(* IEC 61131-3 sources: volt/packages/volt-lsp-iec/test-corpus/pro2193/Device/Plc Logic/Application/09 Misc/Library Manager/L_MC1P_MotionControlBasic (part 4) *)

(* ---- L_MC1P_DRIVESCALING_ENCI900.pou ---- *)
FUNCTION_BLOCK L_MC1P_DRIVESCALING_ENCI900 EXTENDS L_Mc1P_DriveScaling
END_FUNCTION_BLOCK

METHOD CALCACCFACTOR : BOOL
VAR_OUTPUT
	LRSCALEUNITTOACC : LREAL;
	LRSCALEACCTOUNIT : LREAL;
END_VAR
VAR_IN_OUT
	AXIS : _AXIS_REF_REAL;
END_VAR
END_METHOD

METHOD CALCSPEEDFACTOR : BOOL
VAR_OUTPUT
	LRSCALEUNITTOSPEED : LREAL;
	LRSCALESPEEDTOUNIT : LREAL;
END_VAR
VAR_IN_OUT
	AXIS : _AXIS_REF_REAL;
END_VAR
END_METHOD

METHOD CHECKVALIDPOSRESOLUTION : BOOL
VAR_INPUT
	DWPOSRESOLUTION : DWORD;
END_VAR
END_METHOD

METHOD POSDIFFTOSPEEDINC : DINT
VAR_INPUT
	DIPOSDIFF : DINT := 0;
	DWFACTOR : DWORD := 1000;
END_VAR
VAR_IN_OUT
	AXIS : _AXIS_REF_REAL;
END_VAR
END_METHOD

METHOD SPEEDTOPOSDIFFINC : DINT
VAR_INPUT
	DISPEED : DINT := 0;
	DWFACTOR : DWORD := 1000;
END_VAR
VAR_IN_OUT
	AXIS : _AXIS_REF_REAL;
	DIRES : DINT;
END_VAR
END_METHOD

(* ---- L_MC1P_DRIVESCALING_GENERICDRIVE.pou ---- *)
FUNCTION_BLOCK L_MC1P_DRIVESCALING_GENERICDRIVE
VAR_INPUT
	ITFGENERICCONFIG : L_MC1P_IGenericAxisConfiguration;
END_VAR
VAR
	PGENERICAXISCONFIGURATION : POINTER TO L_MC1P_GenericAxisConfiguration;
END_VAR
END_FUNCTION_BLOCK

METHOD CALCACCFACTOR : BOOL
VAR_OUTPUT
	LRSCALEUNITTOACC : LREAL;
	LRSCALEACCTOUNIT : LREAL;
END_VAR
VAR_IN_OUT
	AXIS : _AXIS_REF_REAL;
END_VAR
END_METHOD

METHOD CALCSPEEDFACTOR : BOOL
VAR_OUTPUT
	LRSCALEUNITTOSPEED : LREAL;
	LRSCALESPEEDTOUNIT : LREAL;
END_VAR
VAR_IN_OUT
	AXIS : _AXIS_REF_REAL;
END_VAR
END_METHOD

METHOD CALCTORQUEFACTOR : BOOL
VAR_OUTPUT
	LRSCALETORQUETONORM : LREAL;
	LRSCALETORQUETONORM2 : LREAL;
	LRSCALENORMTOTORQUE : LREAL;
END_VAR
VAR_IN_OUT
	AXIS : _AXIS_REF_REAL;
END_VAR
END_METHOD

METHOD CHECKVALIDPOSRESOLUTION : BOOL
VAR_INPUT
	DWPOSRESOLUTION : DWORD;
END_VAR
END_METHOD

METHOD GETDEFAULTTORQUE : LREAL
VAR_INPUT
	LRREFTORQUE : LREAL;
END_VAR
END_METHOD

METHOD POSDIFFTOSPEEDINC : DINT
VAR_INPUT
	DIPOSDIFF : DINT := 0;
	DWFACTOR : DWORD := 1000;
END_VAR
VAR_IN_OUT
	AXIS : _AXIS_REF_REAL;
END_VAR
END_METHOD

METHOD SPEEDTOPOSDIFFINC : DINT
VAR_INPUT
	DISPEED : DINT := 0;
	DWFACTOR : DWORD := 1000;
END_VAR
VAR_IN_OUT
	AXIS : _AXIS_REF_REAL;
	DIRES : DINT;
END_VAR
END_METHOD

METHOD UPDATEINTERFACE : BOOL
END_METHOD

(* ---- L_MC1P_DRIVESCALING_I500.pou ---- *)
FUNCTION_BLOCK L_MC1P_DRIVESCALING_I500 EXTENDS L_MC1P_DriveScaling
END_FUNCTION_BLOCK

METHOD CALCTORQUEFACTOR : BOOL
VAR_OUTPUT
	LRSCALETORQUETONORM : LREAL;
	LRSCALETORQUETONORM2 : LREAL;
	LRSCALENORMTOTORQUE : LREAL;
END_VAR
VAR_IN_OUT
	AXIS : _AXIS_REF_REAL;
END_VAR
END_METHOD

METHOD GETDEFAULTTORQUE : LREAL
VAR_INPUT
	LRREFTORQUE : LREAL;
END_VAR
END_METHOD

(* ---- L_MC1P_DRIVESCALING_I7XX.pou ---- *)
FUNCTION_BLOCK L_MC1P_DRIVESCALING_I7XX
END_FUNCTION_BLOCK

METHOD CALCACCFACTOR : BOOL
VAR_OUTPUT
	LRSCALEUNITTOACC : LREAL;
	LRSCALEACCTOUNIT : LREAL;
END_VAR
VAR_IN_OUT
	AXIS : _AXIS_REF_REAL;
END_VAR
END_METHOD

METHOD CALCSPEEDFACTOR : BOOL
VAR_OUTPUT
	LRSCALEUNITTOSPEED : LREAL;
	LRSCALESPEEDTOUNIT : LREAL;
END_VAR
VAR_IN_OUT
	AXIS : _AXIS_REF_REAL;
END_VAR
END_METHOD

METHOD CALCTORQUEFACTOR : BOOL
VAR_OUTPUT
	LRSCALETORQUETONORM : LREAL;
	LRSCALETORQUETONORM2 : LREAL;
	LRSCALENORMTOTORQUE : LREAL;
END_VAR
VAR_IN_OUT
	AXIS : _AXIS_REF_REAL;
END_VAR
END_METHOD

METHOD CHECKVALIDPOSRESOLUTION : BOOL
VAR_INPUT
	DWPOSRESOLUTION : DWORD;
END_VAR
END_METHOD

METHOD GETDEFAULTTORQUE : LREAL
VAR_INPUT
	LRREFTORQUE : LREAL;
END_VAR
END_METHOD

METHOD POSDIFFTOSPEEDINC : DINT
VAR_INPUT
	DIPOSDIFF : DINT := 0;
	DWFACTOR : DWORD := 1000;
END_VAR
VAR_IN_OUT
	AXIS : _AXIS_REF_REAL;
END_VAR
END_METHOD

METHOD SPEEDTOPOSDIFFINC : DINT
VAR_INPUT
	DISPEED : DINT := 0;
	DWFACTOR : DWORD := 1000;
END_VAR
VAR_IN_OUT
	AXIS : _AXIS_REF_REAL;
	DIRES : DINT;
END_VAR
END_METHOD

(* ---- L_MC1P_DRIVESPECIFIC_9400HL.pou ---- *)
FUNCTION_BLOCK L_MC1P_DRIVESPECIFIC_9400HL EXTENDS L_MC1P_DriveSpecific_CiA402
VAR
	TPWORKER : L_MC1P_TpWorker_CiA402;
	WSTATESM : WORD;
	DRIVEHOMESTATUSCHANGED : BOOL;
END_VAR
END_FUNCTION_BLOCK

METHOD CALCAFTERREADINPUTS
VAR_IN_OUT
	AXIS : _AXIS_REF_REAL;
END_VAR
END_METHOD

METHOD CALCBEFOREWRITEOUTPUTS
VAR_IN_OUT
	AXIS : _AXIS_REF_REAL;
END_VAR
END_METHOD

METHOD CHECKRESETHOMEPOS
VAR_INPUT
	WFDBSTATUSWORD : WORD;
END_VAR
VAR_IN_OUT
	AXIS : _AXIS_REF_REAL;
END_VAR
END_METHOD

METHOD GETADDITIONALSTATEINFOS : BOOL
VAR_IN_OUT
	AXIS : _AXIS_REF_REAL;
	SCSTATEINFO : L_MC1P_DriveStateCollection;
END_VAR
END_METHOD

METHOD GETCAUSEOFCINH : WORD
VAR_IN_OUT
	AXIS : _AXIS_REF_REAL;
END_VAR
END_METHOD

METHOD GETRECEIVEDATAIMPL : DWORD
VAR_INPUT
	LWMASK : LWORD;
END_VAR
VAR_IN_OUT
	AXIS : _AXIS_REF_REAL;
END_VAR
END_METHOD

METHOD GETSTOACTIVEFROMSTATE : BOOL
VAR_IN_OUT
	AXIS : _AXIS_REF_REAL;
END_VAR
END_METHOD

METHOD HOMECONFIG : BOOL
VAR_INPUT
	LRPOSITION : LREAL;
END_VAR
VAR_OUTPUT
	WINDEX : WORD;
	BYSUBINDEX : BYTE;
	BYNROFBYTE : BYTE;
	DWDATA : DWORD;
	XWRITEPARAM : BOOL;
	XDONE : BOOL;
	XERROR : BOOL;
END_VAR
VAR_IN_OUT
	AXIS : _AXIS_REF_REAL;
	SCHOMEDATA : L_MC1P_HomeParameter;
	WSTEP : WORD;
END_VAR
END_METHOD

METHOD PROZESSCONTROLWORD : BOOL
VAR_IN_OUT
	AXIS : _AXIS_REF_REAL;
END_VAR
END_METHOD

METHOD RECEIVEPARAMETERCALC
VAR_IN_OUT
	AXIS : _AXIS_REF_REAL;
	DATA : ARRAY [1..L_MC1P_Constants.gc_Rec_MaxDataIndex] OF POINTER TO L_MC1P_MappedElement;
END_VAR
END_METHOD

METHOD SETAXISPROPERTIES
VAR_IN_OUT
	AXIS : _AXIS_REF_REAL;
	AXISPROPERTIES : L_MC1P_AxisProperties;
END_VAR
END_METHOD

METHOD SETAXISSTATUSWORD
VAR_IN_OUT
	AXIS : _AXIS_REF_REAL;
	DWAXISSTATUS : DWORD;
END_VAR
END_METHOD

METHOD SETDRIVECONFIGINIT
VAR_IN_OUT
	AXIS : _AXIS_REF_REAL;
END_VAR
END_METHOD

METHOD TRANSMITPARAMETERCALC
VAR_IN_OUT
	AXIS : _AXIS_REF_REAL;
	DATA : ARRAY [1..L_MC1P_Constants.gc_Trans_MaxDataIndex] OF POINTER TO L_MC1P_MappedElement;
END_VAR
END_METHOD

(* ---- L_MC1P_DRIVESPECIFIC_BASIC.pou ---- *)
FUNCTION_BLOCK L_MC1P_DRIVESPECIFIC_BASIC
VAR_INPUT
	XDEFAULTBEHAVIOURASVIRTUAL : BOOL := FALSE;
END_VAR
VAR
	XENABLE : BOOL;
	DIPOS : DINT;
	DIVEL : DINT;
	ITORQUE : INT;
	ITORQUELIMPOS : INT;
	ITORQUELIMNEG : INT;
	DIFOLLOWINGERROR : DINT;
	WERRORCODE : WORD;
	BASICINITERROR : L_IE1P_Error;
	DRIVEHOMESTATUSCHANGED : BOOL;
	DRIVEINITIALIZED : BOOL;
	DRIVEINITIALIZEDERRORREASON : L_IE1P_Error;
	GETITFBRAKE : L_MC1P_IAXIS_REF_BRAKE;
	GETITFCMDBRAKEGRINDIN : L_MC1P_IAxisCommmand;
	GETITFCMDBRAKETEST : L_MC1P_IAxisCommmand;
	HOMESEQUENCESTATE : WORD;
	ITFMOLACCESS : L_MC1P_IMOLAccess;
	ITFPLIACCESS : L_MC1P_IPLIAccess;
	PINSTANCE : POINTER TO BYTE;
END_VAR
END_FUNCTION_BLOCK

METHOD CALCAFTERREADINPUTS
VAR_IN_OUT
	AXIS : _AXIS_REF_REAL;
END_VAR
END_METHOD

METHOD CALCBEFOREREADINPUTS
VAR_IN_OUT
	AXIS : _AXIS_REF_REAL;
END_VAR
END_METHOD

METHOD CALCBEFOREWRITEOUTPUTS
VAR_IN_OUT
	AXIS : _AXIS_REF_REAL;
END_VAR
END_METHOD

METHOD CHECKAVAILABLECONTROLMODE : BOOL
VAR_IN_OUT
	AXIS : _AXIS_REF_REAL;
	POSCTRLDRIVEAVAILABLE : L_IE1P_Error;
	POSCTRLPLCAVAILABLE : L_IE1P_Error;
	SPEEDCTRLDRIVEAVAILABLE : L_IE1P_Error;
	TORQUECTRLDRIVE : L_IE1P_Error;
END_VAR
END_METHOD

METHOD CHECKRESETHOMEPOS
VAR_INPUT
	WFDBSTATUSWORD : WORD;
END_VAR
VAR_IN_OUT
	AXIS : _AXIS_REF_REAL;
END_VAR
END_METHOD

METHOD CHECKSAFETYOPTIONAVAILABLE : BOOL
VAR_INPUT
	DWPRODUCTCODE : DWORD;
END_VAR
END_METHOD

METHOD COLLECTDRIVESTATE : BOOL
VAR_IN_OUT
	AXIS : _AXIS_REF_REAL;
	SCSTATEINFO : L_MC1P_DriveStateCollection;
END_VAR
END_METHOD

METHOD CONTROLDRIVE : BOOL
VAR_INPUT
	XENABLE : BOOL;
END_VAR
VAR_IN_OUT
	AXIS : _AXIS_REF_REAL;
END_VAR
END_METHOD

METHOD DRIVECONFIGDATA
VAR_INPUT
	PCONFIGINFO : POINTER TO L_MC1P_AdditionalConfigInfo;
END_VAR
VAR_IN_OUT
	AXIS : _AXIS_REF_REAL;
END_VAR
END_METHOD

METHOD DRIVEFAULTSTATUS : BOOL
VAR_IN_OUT
	AXIS : _AXIS_REF_REAL;
	SCSTATEINFO : L_MC1P_DriveStateCollection;
END_VAR
END_METHOD

METHOD GETBRAKE : POINTER TO L_MC1P_BrakeControlBase
VAR_IN_OUT
	AXIS : _AXIS_REF_REAL;
END_VAR
END_METHOD

METHOD GETBRAKESERVICE : POINTER TO L_MC1P_BrakeService
VAR_IN_OUT
	AXIS : _AXIS_REF_REAL;
END_VAR
END_METHOD

METHOD GETCAUSEOFCINH : WORD
VAR_IN_OUT
	AXIS : _AXIS_REF_REAL;
END_VAR
END_METHOD

METHOD GETFDBSTATUSWORD : WORD
VAR_IN_OUT
	AXIS : _AXIS_REF_REAL;
END_VAR
END_METHOD

METHOD GETIECADRESS : BOOL
VAR_IN_OUT
	AXIS : _AXIS_REF_REAL;
	M_PPDOINFOCONNECTOR : POINTER TO IoConfigConnector;
	ATRANSELEMENT : ARRAY [1.._AXIS_REF_REAL.c_wMaxTransElem] OF L_MC1P_MappedElement;
	WTRANSELEMENTS : WORD;
	LWTRANSDATA : LWORD;
	LWRECDATA : LWORD;
	WRECEIVEELEMENTS : WORD;
	ARECEIVEELEMENT : ARRAY [1.._AXIS_REF_REAL.c_wMaxRecElem] OF L_MC1P_MappedElement;
END_VAR
END_METHOD

METHOD GETOPTIONALACTVEL : BOOL
VAR_IN_OUT
	LRVEL : LREAL;
END_VAR
END_METHOD

METHOD GETRECEIVEDATAIMPL : DWORD
VAR_INPUT
	LWMASK : LWORD;
END_VAR
VAR_IN_OUT
	AXIS : _AXIS_REF_REAL;
END_VAR
END_METHOD

METHOD GETSTATUSWORDS
VAR_OUTPUT
	STATUSWORD1 : WORD;
	STATUSWORD2 : WORD;
	STATUSWORD3 : WORD;
	STATUSWORD4 : WORD;
END_VAR
VAR_IN_OUT
	AXIS : _AXIS_REF_REAL;
END_VAR
END_METHOD

METHOD GETTRANSMITDATAIMPL : DWORD
VAR_INPUT
	LWMASK : LWORD;
END_VAR
VAR_IN_OUT
	AXIS : _AXIS_REF_REAL;
END_VAR
END_METHOD

METHOD GETTRANSMITDATALREALIMPL : LREAL
VAR_INPUT
	LWMASK : LWORD;
END_VAR
VAR_IN_OUT
	AXIS : _AXIS_REF_REAL;
END_VAR
END_METHOD

METHOD HOMECONFIG : BOOL
VAR_INPUT
	LRPOSITION : LREAL;
END_VAR
VAR_OUTPUT
	WINDEX : WORD;
	BYSUBINDEX : BYTE;
	BYNROFBYTE : BYTE;
	DWDATA : DWORD;
	XWRITEPARAM : BOOL;
	XDONE : BOOL;
	XERROR : BOOL;
END_VAR
VAR_IN_OUT
	AXIS : _AXIS_REF_REAL;
	SCHOMEDATA : L_MC1P_HomeParameter;
	WSTEP : WORD;
END_VAR
END_METHOD

METHOD HOMEPOSPERMANENTSETACTIVE : BOOL
VAR_IN_OUT
	AXIS : _AXIS_REF_REAL;
END_VAR
END_METHOD

METHOD RECEIVEPARAMETER
VAR_INPUT
	WPARAMETER : WORD;
	PADRESS : POINTER TO BYTE;
	WSIZE : WORD;
END_VAR
VAR_IN_OUT
	AXIS : _AXIS_REF_REAL;
END_VAR
END_METHOD

METHOD RECEIVEPARAMETERCALC
VAR_IN_OUT
	AXIS : _AXIS_REF_REAL;
	DATA : ARRAY [1..L_MC1P_Constants.gc_Rec_MaxDataIndex] OF POINTER TO L_MC1P_MappedElement;
END_VAR
END_METHOD

METHOD RESETDRIVECONTROL
VAR_INPUT
	XRESETDRIVEERROR : BOOL;
END_VAR
END_METHOD

METHOD RESTOREADDITIONALRETAINDATA
VAR_INPUT
	PDATA : POINTER TO L_MC1P_uRetainData;
END_VAR
END_METHOD

METHOD SETAXISPROPERTIES
VAR_IN_OUT
	AXIS : _AXIS_REF_REAL;
	AXISPROPERTIES : L_MC1P_AxisProperties;
END_VAR
END_METHOD

METHOD SETAXISSTATUSWORD
VAR_IN_OUT
	AXIS : _AXIS_REF_REAL;
	DWAXISSTATUS : DWORD;
END_VAR
END_METHOD

METHOD SETBASICINITIALISATION
VAR_IN_OUT
	AXIS : _AXIS_REF_REAL;
END_VAR
END_METHOD

METHOD SETCONTROLWORDS
VAR_INPUT
	CONTROLWORD1 : WORD;
	CONTROLWORD2 : WORD;
	CONTROLWORD3 : WORD;
	CONTROLWORD4 : WORD;
END_VAR
VAR_IN_OUT
	AXIS : _AXIS_REF_REAL;
END_VAR
END_METHOD

METHOD SETDCBRAKE
VAR_INPUT
	XSETDCBRAKE : BOOL;
END_VAR
VAR_OUTPUT
	XDCBRAKEACTIVE : BOOL;
END_VAR
VAR_IN_OUT
	AXIS : _AXIS_REF_REAL;
END_VAR
END_METHOD

METHOD SETDRIVECONFIG
VAR_OUTPUT
	XDONE : BOOL;
	XERROR : BOOL;
	WERRORID : WORD;
END_VAR
VAR_IN_OUT
	AXIS : _AXIS_REF_REAL;
END_VAR
END_METHOD

METHOD SETDRIVECONFIGINIT
VAR_IN_OUT
	AXIS : _AXIS_REF_REAL;
END_VAR
END_METHOD

METHOD SETSPEEDCTRLLIMITATION : BOOL
VAR_INPUT
	XLIMIT : BOOL;
END_VAR
VAR_IN_OUT
	AXIS : _AXIS_REF_REAL;
END_VAR
END_METHOD

METHOD SETSPEEDCTRLLOADVALUE
VAR_INPUT
	XLOAD : BOOL;
	LRVALUE : LREAL;
END_VAR
VAR_IN_OUT
	AXIS : _AXIS_REF_REAL;
END_VAR
END_METHOD

METHOD STOREADDITIONALRETAINDATA
VAR_INPUT
	PDATA : POINTER TO L_MC1P_uRetainData;
END_VAR
END_METHOD

METHOD TRANSMITPARAMETER
VAR_INPUT
	WPARAMETER : WORD;
	PADRESS : POINTER TO BYTE;
	WSIZE : WORD;
END_VAR
VAR_IN_OUT
	AXIS : _AXIS_REF_REAL;
END_VAR
END_METHOD

METHOD TRANSMITPARAMETERCALC
VAR_IN_OUT
	AXIS : _AXIS_REF_REAL;
	DATA : ARRAY [1..L_MC1P_Constants.gc_Trans_MaxDataIndex] OF POINTER TO L_MC1P_MappedElement;
END_VAR
END_METHOD

METHOD UPDATEMAPPING
VAR_INPUT
	PTASKMAPLIST : POINTER TO IoStandard.IoConfigTaskMap;
	NCOUNT : DINT;
	PPDOINFOCONNECTOR : POINTER TO IoConfigConnector;
END_VAR
VAR_IN_OUT
	AXIS : _AXIS_REF_REAL;
END_VAR
END_METHOD

(* ---- L_MC1P_DRIVESPECIFIC_CIA402.pou ---- *)
FUNCTION_BLOCK L_MC1P_DRIVESPECIFIC_CIA402
VAR_INPUT
	WOFFSETDRIVEPARA : WORD;
END_VAR
VAR
	ECONTROLMODEDRIVE : SINT := 0;
	XUSEIPMODENOTCSP : BOOL := FALSE;
	XUSEVLMODENOTCSV : BOOL := FALSE;
	CIA_CTRL : WORD;
	CIA_OPMOD : SINT;
	CIA_STATE : WORD;
	CIA_OPMODACT : SINT;
	CIA_VLACTVELOCITY : INT;
	CIA_VLTARGETVELOCITY : INT;
	CIA_STATEOLD : WORD;
	WHOMESTATE : WORD;
	REFCIA_CTRL : REFERENCE TO WORD;
	REFCIA_OPMOD : REFERENCE TO SINT;
	REFCIA_STATE : REFERENCE TO WORD;
	REFCIA_OPMODACT : REFERENCE TO SINT;
	DWSAFETYCONTROL : DWORD;
	DWSAFETYSTATE : DWORD;
	DWSAFETYIOSTATE : DWORD;
	WLENZEEXTSTATUSWORD : WORD := 0;
	XTEXTREFID603FSUPPORTED : BOOL;
	WTEXTREFID603F : WORD;
	WTEXTREFID_SLAVE : WORD;
	LRDECTIME : LREAL;
	XQSPRAMPEND : BOOL;
	BASICINITERROR : L_IE1P_Types.L_IE1P_Error;
	DRIVEHOMESTATUSCHANGED : BOOL;
	DRIVEINITIALIZED : BOOL;
	DRIVEINITIALIZEDERRORREASON : L_IE1P_Types.L_IE1P_Error;
	GETITFBRAKE : L_MC1P_IAXIS_REF_BRAKE;
	GETITFCMDBRAKEGRINDIN : L_MC1P_IAxisCommmand;
	GETITFCMDBRAKETEST : L_MC1P_IAxisCommmand;
	HOMESEQUENCESTATE : WORD;
	ITFMOLACCESS : L_MC1P_IMOLAccess;
	ITFPLIACCESS : L_MC1P_IPLIAccess;
	PINSTANCE : POINTER TO BYTE;
END_VAR
END_FUNCTION_BLOCK

METHOD CALCAFTERCIA402STM : BOOL
VAR_IN_OUT
	AXIS : _AXIS_REF_REAL;
END_VAR
END_METHOD

METHOD GETADDITIONALSTATEINFOS : BOOL
VAR_IN_OUT
	AXIS : _AXIS_REF_REAL;
	SCSTATEINFO : L_MC1P_DriveStateCollection;
END_VAR
END_METHOD

METHOD GETDRIVEQSPDONE : BOOL
VAR_IN_OUT
	AXIS : _AXIS_REF_REAL;
	SCSTATEINFO : L_MC1P_DriveStateCollection;
END_VAR
END_METHOD

METHOD GETINTCONTROLMODE : SINT
VAR_INPUT
	ECONTROLMODE : L_MC1P_ControlMode;
END_VAR
VAR_IN_OUT
	AXIS : _AXIS_REF_REAL;
END_VAR
END_METHOD

METHOD GETSTOACTIVEFROMSTATE : BOOL
VAR_IN_OUT
	AXIS : _AXIS_REF_REAL;
END_VAR
END_METHOD

METHOD GETTEXTREFIDFROMERRORCODE : WORD
VAR_INPUT
	DWERRORID : DWORD;
END_VAR
VAR_IN_OUT
	AXIS : _AXIS_REF_REAL;
END_VAR
END_METHOD

METHOD GETTEXTREFIDFROMTABLE : BOOL
VAR_INPUT
	DWERRORID : DWORD;
	XSAFETYDEVICE : BOOL;
END_VAR
VAR_IN_OUT
	WTEXTREFID : WORD;
END_VAR
END_METHOD

METHOD HOMESEQUENCE
VAR_IN_OUT
	AXIS : _AXIS_REF_REAL;
END_VAR
END_METHOD

METHOD PROZESSCONTROLWORD : BOOL
VAR_IN_OUT
	AXIS : _AXIS_REF_REAL;
END_VAR
END_METHOD

METHOD SERVICEMODEHANDLINGINDRIVEACTIVE : BOOL
END_METHOD

METHOD FB_INIT : BOOL
VAR_INPUT
	BINITRETAINS : BOOL;
	BINCOPYCODE : BOOL;
END_VAR
END_METHOD

METHOD CALCAFTERREADINPUTS
VAR_IN_OUT
	AXIS : _AXIS_REF_REAL;
END_VAR
END_METHOD

METHOD CALCBEFOREREADINPUTS
VAR_IN_OUT
	AXIS : _AXIS_REF_REAL;
END_VAR
END_METHOD

METHOD CALCBEFOREWRITEOUTPUTS
VAR_IN_OUT
	AXIS : _AXIS_REF_REAL;
END_VAR
END_METHOD

METHOD CHECKAVAILABLECONTROLMODE : BOOL
VAR_IN_OUT
	AXIS : _AXIS_REF_REAL;
	POSCTRLDRIVEAVAILABLE : L_IE1P_Types.L_IE1P_Error;
	POSCTRLPLCAVAILABLE : L_IE1P_Types.L_IE1P_Error;
	SPEEDCTRLDRIVEAVAILABLE : L_IE1P_Types.L_IE1P_Error;
	TORQUECTRLDRIVE : L_IE1P_Types.L_IE1P_Error;
END_VAR
END_METHOD

METHOD CHECKRESETHOMEPOS
VAR_INPUT
	WFDBSTATUSWORD : WORD;
END_VAR
VAR_IN_OUT
	AXIS : _AXIS_REF_REAL;
END_VAR
END_METHOD

METHOD CHECKSAFETYOPTIONAVAILABLE : BOOL
VAR_INPUT
	DWPRODUCTCODE : DWORD;
END_VAR
END_METHOD

METHOD COLLECTDRIVESTATE : BOOL
VAR_IN_OUT
	AXIS : _AXIS_REF_REAL;
	SCSTATEINFO : L_MC1P_DriveStateCollection;
END_VAR
END_METHOD

METHOD CONTROLDRIVE : BOOL
VAR_INPUT
	XENABLE : BOOL;
END_VAR
VAR_IN_OUT
	AXIS : _AXIS_REF_REAL;
END_VAR
END_METHOD

METHOD DRIVECONFIGDATA
VAR_INPUT
	PCONFIGINFO : POINTER TO L_MC1P_AdditionalConfigInfo;
END_VAR
VAR_IN_OUT
	AXIS : _AXIS_REF_REAL;
END_VAR
END_METHOD

METHOD DRIVEFAULTSTATUS : BOOL
VAR_IN_OUT
	AXIS : _AXIS_REF_REAL;
	SCSTATEINFO : L_MC1P_DriveStateCollection;
END_VAR
END_METHOD

METHOD GETBRAKE : POINTER TO L_MC1P_BrakeControlBase
VAR_IN_OUT
	AXIS : _AXIS_REF_REAL;
END_VAR
END_METHOD

METHOD GETBRAKESERVICE : POINTER TO L_MC1P_BrakeService
VAR_IN_OUT
	AXIS : _AXIS_REF_REAL;
END_VAR
END_METHOD

METHOD GETCAUSEOFCINH : WORD
VAR_IN_OUT
	AXIS : _AXIS_REF_REAL;
END_VAR
END_METHOD

METHOD GETFDBSTATUSWORD : WORD
VAR_IN_OUT
	AXIS : _AXIS_REF_REAL;
END_VAR
END_METHOD

METHOD GETIECADRESS : BOOL
VAR_IN_OUT
	AXIS : _AXIS_REF_REAL;
	M_PPDOINFOCONNECTOR : POINTER TO IoStandard.IoConfigConnector;
	ATRANSELEMENT : ARRAY [1..._AXIS_REF_REAL.c_wMaxTransElem] OF L_MC1P_MappedElement;
	WTRANSELEMENTS : WORD;
	LWTRANSDATA : LWORD;
	LWRECDATA : LWORD;
	WRECEIVEELEMENTS : WORD;
	ARECEIVEELEMENT : ARRAY [1..._AXIS_REF_REAL.c_wMaxRecElem] OF L_MC1P_MappedElement;
END_VAR
END_METHOD

METHOD GETOPTIONALACTVEL : BOOL
VAR_IN_OUT
	LRVEL : LREAL;
END_VAR
END_METHOD

METHOD GETRECEIVEDATAIMPL : DWORD
VAR_INPUT
	LWMASK : LWORD;
END_VAR
VAR_IN_OUT
	AXIS : _AXIS_REF_REAL;
END_VAR
END_METHOD

METHOD GETSTATUSWORDS
VAR_OUTPUT
	STATUSWORD1 : WORD;
	STATUSWORD2 : WORD;
	STATUSWORD3 : WORD;
	STATUSWORD4 : WORD;
END_VAR
VAR_IN_OUT
	AXIS : _AXIS_REF_REAL;
END_VAR
END_METHOD

METHOD GETTRANSMITDATAIMPL : DWORD
VAR_INPUT
	LWMASK : LWORD;
END_VAR
VAR_IN_OUT
	AXIS : _AXIS_REF_REAL;
END_VAR
END_METHOD

METHOD GETTRANSMITDATALREALIMPL : LREAL
VAR_INPUT
	LWMASK : LWORD;
END_VAR
VAR_IN_OUT
	AXIS : _AXIS_REF_REAL;
END_VAR
END_METHOD

METHOD HOMECONFIG : BOOL
VAR_INPUT
	LRPOSITION : LREAL;
END_VAR
VAR_OUTPUT
	WINDEX : WORD;
	BYSUBINDEX : BYTE;
	BYNROFBYTE : BYTE;
	DWDATA : DWORD;
	XWRITEPARAM : BOOL;
	XDONE : BOOL;
	XERROR : BOOL;
END_VAR
VAR_IN_OUT
	AXIS : _AXIS_REF_REAL;
	SCHOMEDATA : L_MC1P_HomeParameter;
	WSTEP : WORD;
END_VAR
END_METHOD

METHOD HOMEPOSPERMANENTSETACTIVE : BOOL
VAR_IN_OUT
	AXIS : _AXIS_REF_REAL;
END_VAR
END_METHOD

METHOD RECEIVEPARAMETERCALC
VAR_IN_OUT
	AXIS : _AXIS_REF_REAL;
	DATA : ARRAY [1..L_MC1P_Constants.gc_Rec_MaxDataIndex] OF POINTER TO L_MC1P_MappedElement;
END_VAR
END_METHOD

METHOD RECEIVEPARAMETER
VAR_INPUT
	WPARAMETER : WORD;
	PADRESS : POINTER TO BYTE;
	WSIZE : WORD;
END_VAR
VAR_IN_OUT
	AXIS : _AXIS_REF_REAL;
END_VAR
END_METHOD

METHOD RESETDRIVECONTROL
VAR_INPUT
	XRESETDRIVEERROR : BOOL;
END_VAR
END_METHOD

METHOD RESTOREADDITIONALRETAINDATA
VAR_INPUT
	PDATA : POINTER TO L_MC1P_uRetainData;
END_VAR
END_METHOD

METHOD SETAXISPROPERTIES
VAR_IN_OUT
	AXIS : _AXIS_REF_REAL;
	AXISPROPERTIES : L_MC1P_AxisProperties;
END_VAR
END_METHOD

METHOD SETAXISSTATUSWORD
VAR_IN_OUT
	AXIS : _AXIS_REF_REAL;
	DWAXISSTATUS : DWORD;
END_VAR
END_METHOD

METHOD SETBASICINITIALISATION
VAR_IN_OUT
	AXIS : _AXIS_REF_REAL;
END_VAR
END_METHOD

METHOD SETCONTROLWORDS
VAR_INPUT
	CONTROLWORD1 : WORD;
	CONTROLWORD2 : WORD;
	CONTROLWORD3 : WORD;
	CONTROLWORD4 : WORD;
END_VAR
VAR_IN_OUT
	AXIS : _AXIS_REF_REAL;
END_VAR
END_METHOD

METHOD SETDCBRAKE
VAR_INPUT
	XSETDCBRAKE : BOOL;
END_VAR
VAR_OUTPUT
	XDCBRAKEACTIVE : BOOL;
END_VAR
VAR_IN_OUT
	AXIS : _AXIS_REF_REAL;
END_VAR
END_METHOD

METHOD SETDRIVECONFIGINIT
VAR_IN_OUT
	AXIS : _AXIS_REF_REAL;
END_VAR
END_METHOD

METHOD SETSPEEDCTRLLIMITATION : BOOL
VAR_INPUT
	XLIMIT : BOOL;
END_VAR
VAR_IN_OUT
	AXIS : _AXIS_REF_REAL;
END_VAR
END_METHOD

METHOD SETSPEEDCTRLLOADVALUE
VAR_INPUT
	XLOAD : BOOL;
	LRVALUE : LREAL;
END_VAR
VAR_IN_OUT
	AXIS : _AXIS_REF_REAL;
END_VAR
END_METHOD

METHOD STOREADDITIONALRETAINDATA
VAR_INPUT
	PDATA : POINTER TO L_MC1P_uRetainData;
END_VAR
END_METHOD

METHOD TRANSMITPARAMETERCALC
VAR_IN_OUT
	AXIS : _AXIS_REF_REAL;
	DATA : ARRAY [1..L_MC1P_Constants.gc_Trans_MaxDataIndex] OF POINTER TO L_MC1P_MappedElement;
END_VAR
END_METHOD

METHOD TRANSMITPARAMETER
VAR_INPUT
	WPARAMETER : WORD;
	PADRESS : POINTER TO BYTE;
	WSIZE : WORD;
END_VAR
VAR_IN_OUT
	AXIS : _AXIS_REF_REAL;
END_VAR
END_METHOD

METHOD UPDATEMAPPING
VAR_INPUT
	PTASKMAPLIST : POINTER TO IoStandard.IoConfigTaskMap;
	NCOUNT : DINT;
	PPDOINFOCONNECTOR : POINTER TO IoStandard.IoConfigConnector;
END_VAR
VAR_IN_OUT
	AXIS : _AXIS_REF_REAL;
END_VAR
END_METHOD

(* ---- L_MC1P_DRIVESPECIFIC_ENC.pou ---- *)
FUNCTION_BLOCK L_MC1P_DRIVESPECIFIC_ENC
VAR
	BASICINITERROR : L_IE1P_Error;
	DRIVEHOMESTATUSCHANGED : BOOL;
	DRIVEINITIALIZED : BOOL;
	DRIVEINITIALIZEDERRORREASON : L_IE1P_Error;
	GETITFBRAKE : L_MC1P_IAXIS_REF_BRAKE;
	GETITFCMDBRAKEGRINDIN : L_MC1P_IAxisCommmand;
	GETITFCMDBRAKETEST : L_MC1P_IAxisCommmand;
	HOMESEQUENCESTATE : WORD;
	ITFMOLACCESS : L_MC1P_IMOLAccess;
	ITFPLIACCESS : L_MC1P_IPLIAccess;
	PINSTANCE : POINTER TO BYTE;
END_VAR
END_FUNCTION_BLOCK

METHOD CALCAFTERREADINPUTS
VAR_IN_OUT
	AXIS : _AXIS_REF_REAL;
END_VAR
END_METHOD

METHOD CALCBEFOREREADINPUTS
VAR_IN_OUT
	AXIS : _AXIS_REF_REAL;
END_VAR
END_METHOD

METHOD CALCBEFOREWRITEOUTPUTS
VAR_IN_OUT
	AXIS : _AXIS_REF_REAL;
END_VAR
END_METHOD

METHOD CHECKAVAILABLECONTROLMODE : BOOL
VAR_IN_OUT
	AXIS : _AXIS_REF_REAL;
	POSCTRLDRIVEAVAILABLE : L_IE1P_Error;
	POSCTRLPLCAVAILABLE : L_IE1P_Error;
	SPEEDCTRLDRIVEAVAILABLE : L_IE1P_Error;
	TORQUECTRLDRIVE : L_IE1P_Error;
END_VAR
END_METHOD

METHOD CHECKRESETHOMEPOS
VAR_INPUT
	WFDBSTATUSWORD : WORD;
END_VAR
VAR_IN_OUT
	AXIS : _AXIS_REF_REAL;
END_VAR
END_METHOD

METHOD CHECKSAFETYOPTIONAVAILABLE : BOOL
VAR_INPUT
	DWPRODUCTCODE : DWORD;
END_VAR
END_METHOD

METHOD COLLECTDRIVESTATE : BOOL
VAR_IN_OUT
	AXIS : _AXIS_REF_REAL;
	SCSTATEINFO : L_MC1P_DriveStateCollection;
END_VAR
END_METHOD

METHOD CONTROLDRIVE : BOOL
VAR_INPUT
	XENABLE : BOOL;
END_VAR
VAR_IN_OUT
	AXIS : _AXIS_REF_REAL;
END_VAR
END_METHOD

METHOD DRIVECONFIGDATA
VAR_INPUT
	PCONFIGINFO : POINTER TO L_MC1P_AdditionalConfigInfo;
END_VAR
VAR_IN_OUT
	AXIS : _AXIS_REF_REAL;
END_VAR
END_METHOD

METHOD DRIVEFAULTSTATUS : BOOL
VAR_IN_OUT
	AXIS : _AXIS_REF_REAL;
	SCSTATEINFO : L_MC1P_DriveStateCollection;
END_VAR
END_METHOD

METHOD GETBRAKE : POINTER TO L_MC1P_BrakeControlBase
VAR_IN_OUT
	AXIS : _AXIS_REF_REAL;
END_VAR
END_METHOD

METHOD GETBRAKESERVICE : POINTER TO L_MC1P_BrakeService
VAR_IN_OUT
	AXIS : _AXIS_REF_REAL;
END_VAR
END_METHOD

METHOD GETCAUSEOFCINH : WORD
VAR_IN_OUT
	AXIS : _AXIS_REF_REAL;
END_VAR
END_METHOD

METHOD GETFDBSTATUSWORD : WORD
VAR_IN_OUT
	AXIS : _AXIS_REF_REAL;
END_VAR
END_METHOD

METHOD GETIECADRESS : BOOL
VAR_IN_OUT
	AXIS : _AXIS_REF_REAL;
	M_PPDOINFOCONNECTOR : POINTER TO IoConfigConnector;
	ATRANSELEMENT : ARRAY [1.._AXIS_REF_REAL.c_wMaxTransElem] OF L_MC1P_MappedElement;
	WTRANSELEMENTS : WORD;
	LWTRANSDATA : LWORD;
	LWRECDATA : LWORD;
	WRECEIVEELEMENTS : WORD;
	ARECEIVEELEMENT : ARRAY [1.._AXIS_REF_REAL.c_wMaxRecElem] OF L_MC1P_MappedElement;
END_VAR
END_METHOD

METHOD GETOPTIONALACTVEL : BOOL
VAR_IN_OUT
	LRVEL : LREAL;
END_VAR
END_METHOD

METHOD GETRECEIVEDATAIMPL : DWORD
VAR_INPUT
	LWMASK : LWORD;
END_VAR
VAR_IN_OUT
	AXIS : _AXIS_REF_REAL;
END_VAR
END_METHOD

METHOD GETSTATUSWORDS
VAR_OUTPUT
	STATUSWORD1 : WORD;
	STATUSWORD2 : WORD;
	STATUSWORD3 : WORD;
	STATUSWORD4 : WORD;
END_VAR
VAR_IN_OUT
	AXIS : _AXIS_REF_REAL;
END_VAR
END_METHOD

METHOD GETTRANSMITDATAIMPL : DWORD
VAR_INPUT
	LWMASK : LWORD;
END_VAR
VAR_IN_OUT
	AXIS : _AXIS_REF_REAL;
END_VAR
END_METHOD

METHOD GETTRANSMITDATALREALIMPL : LREAL
VAR_INPUT
	LWMASK : LWORD;
END_VAR
VAR_IN_OUT
	AXIS : _AXIS_REF_REAL;
END_VAR
END_METHOD

METHOD HOMECONFIG : BOOL
VAR_INPUT
	LRPOSITION : LREAL;
END_VAR
VAR_OUTPUT
	WINDEX : WORD;
	BYSUBINDEX : BYTE;
	BYNROFBYTE : BYTE;
	DWDATA : DWORD;
	XWRITEPARAM : BOOL;
	XDONE : BOOL;
	XERROR : BOOL;
END_VAR
VAR_IN_OUT
	AXIS : _AXIS_REF_REAL;
	SCHOMEDATA : L_MC1P_HomeParameter;
	WSTEP : WORD;
END_VAR
END_METHOD

METHOD HOMEPOSPERMANENTSETACTIVE : BOOL
VAR_IN_OUT
	AXIS : _AXIS_REF_REAL;
END_VAR
END_METHOD

METHOD RECEIVEPARAMETER
VAR_INPUT
	WPARAMETER : WORD;
	PADRESS : POINTER TO BYTE;
	WSIZE : WORD;
END_VAR
VAR_IN_OUT
	AXIS : _AXIS_REF_REAL;
END_VAR
END_METHOD

METHOD RECEIVEPARAMETERCALC
VAR_IN_OUT
	AXIS : _AXIS_REF_REAL;
	DATA : ARRAY [1..L_MC1P_Constants.gc_Rec_MaxDataIndex] OF POINTER TO L_MC1P_MappedElement;
END_VAR
END_METHOD

METHOD RESETDRIVECONTROL
VAR_INPUT
	XRESETDRIVEERROR : BOOL;
END_VAR
END_METHOD

METHOD RESTOREADDITIONALRETAINDATA
VAR_INPUT
	PDATA : POINTER TO L_MC1P_uRetainData;
END_VAR
END_METHOD

METHOD SETAXISPROPERTIES
VAR_IN_OUT
	AXIS : _AXIS_REF_REAL;
	AXISPROPERTIES : L_MC1P_AxisProperties;
END_VAR
END_METHOD

METHOD SETAXISSTATUSWORD
VAR_IN_OUT
	AXIS : _AXIS_REF_REAL;
	DWAXISSTATUS : DWORD;
END_VAR
END_METHOD

METHOD SETBASICINITIALISATION
VAR_IN_OUT
	AXIS : _AXIS_REF_REAL;
END_VAR
END_METHOD

METHOD SETCONTROLWORDS
VAR_INPUT
	CONTROLWORD1 : WORD;
	CONTROLWORD2 : WORD;
	CONTROLWORD3 : WORD;
	CONTROLWORD4 : WORD;
END_VAR
VAR_IN_OUT
	AXIS : _AXIS_REF_REAL;
END_VAR
END_METHOD

METHOD SETDCBRAKE
VAR_INPUT
	XSETDCBRAKE : BOOL;
END_VAR
VAR_OUTPUT
	XDCBRAKEACTIVE : BOOL;
END_VAR
VAR_IN_OUT
	AXIS : _AXIS_REF_REAL;
END_VAR
END_METHOD

METHOD SETDRIVECONFIG
VAR_OUTPUT
	XDONE : BOOL;
	XERROR : BOOL;
	WERRORID : WORD;
END_VAR
VAR_IN_OUT
	AXIS : _AXIS_REF_REAL;
END_VAR
END_METHOD

METHOD SETDRIVECONFIGINIT
VAR_IN_OUT
	AXIS : _AXIS_REF_REAL;
END_VAR
END_METHOD

METHOD SETSPEEDCTRLLIMITATION : BOOL
VAR_INPUT
	XLIMIT : BOOL;
END_VAR
VAR_IN_OUT
	AXIS : _AXIS_REF_REAL;
END_VAR
END_METHOD

METHOD SETSPEEDCTRLLOADVALUE
VAR_INPUT
	XLOAD : BOOL;
	LRVALUE : LREAL;
END_VAR
VAR_IN_OUT
	AXIS : _AXIS_REF_REAL;
END_VAR
END_METHOD

METHOD STOREADDITIONALRETAINDATA
VAR_INPUT
	PDATA : POINTER TO L_MC1P_uRetainData;
END_VAR
END_METHOD

METHOD TRANSMITPARAMETER
VAR_INPUT
	WPARAMETER : WORD;
	PADRESS : POINTER TO BYTE;
	WSIZE : WORD;
END_VAR
VAR_IN_OUT
	AXIS : _AXIS_REF_REAL;
END_VAR
END_METHOD

METHOD TRANSMITPARAMETERCALC
VAR_IN_OUT
	AXIS : _AXIS_REF_REAL;
	DATA : ARRAY [1..L_MC1P_Constants.gc_Trans_MaxDataIndex] OF POINTER TO L_MC1P_MappedElement;
END_VAR
END_METHOD

METHOD UPDATEMAPPING
VAR_INPUT
	PTASKMAPLIST : POINTER TO IoStandard.IoConfigTaskMap;
	NCOUNT : DINT;
	PPDOINFOCONNECTOR : POINTER TO IoConfigConnector;
END_VAR
VAR_IN_OUT
	AXIS : _AXIS_REF_REAL;
END_VAR
END_METHOD

(* ---- L_MC1P_DRIVESPECIFIC_ENC_BPB.pou ---- *)
FUNCTION_BLOCK L_MC1P_DRIVESPECIFIC_ENC_BPB EXTENDS L_MC1P_DriveSpecific_ENC
VAR
	PDWCOUNTER : POINTER TO DWORD := 0;
	PWMICSECTICK : POINTER TO WORD := 0;
	WINDEX1027H_VALUE : WORD;
	XMAPPINGDONE : BOOL;
	CONST_MAX_COUNTER : BYTE := 2;
	CONST_ID_EPM_S600 : WORD := 16#991;
	CONST_ID_EPM_S601 : WORD := 16#993;
	CONST_ID_EPM_S602 : WORD := 16#992;
	CONST_ID_EPM_S603 : WORD := 16#994;
	CONST_ID_EPM_S604 : WORD := 16#995;
	CONST_EPM_600_CNT_VALUE_PARID : DWORD := 1001;
	CONST_EPM_600_TICK_PARID : DWORD := 1004;
	CONST_EPM_601_CNT1_VALUE_PARID : DWORD := 1001;
	CONST_EPM_601_CNT2_VALUE_PARID : DWORD := 1002;
	CONST_EPM_602_CNT_VALUE_PARID : DWORD := 1001;
	CONST_EPM_602_TICK_PARID : DWORD := 1003;
	CONST_EPM_603_CNT1_VALUE_PARID : DWORD := 1001;
	CONST_EPM_603_CNT2_VALUE_PARID : DWORD := 1002;
	CONST_EPM_604_CNT_VALUE_PARID : DWORD := 1001;
	CONST_EPM_604_TICK_PARID : DWORD := 1002;
	BASICINITERROR : L_IE1P_Error;
	DRIVEINITIALIZED : BOOL;
	DRIVEINITIALIZEDERRORREASON : L_IE1P_Error;
END_VAR
END_FUNCTION_BLOCK

METHOD GETIECADRESS : BOOL
VAR_IN_OUT
	AXIS : _AXIS_REF_REAL;
	M_PPDOINFOCONNECTOR : POINTER TO IoConfigConnector;
	ATRANSELEMENT : ARRAY [1.._AXIS_REF_REAL.c_wMaxTransElem] OF L_MC1P_MappedElement;
	WTRANSELEMENTS : WORD;
	LWTRANSDATA : LWORD;
	LWRECDATA : LWORD;
	WRECEIVEELEMENTS : WORD;
	ARECEIVEELEMENT : ARRAY [1.._AXIS_REF_REAL.c_wMaxRecElem] OF L_MC1P_MappedElement;
END_VAR
END_METHOD

METHOD RECEIVEPARAMETERCALC
VAR_IN_OUT
	AXIS : _AXIS_REF_REAL;
	DATA : ARRAY [1..L_MC1P_Constants.gc_Rec_MaxDataIndex] OF POINTER TO L_MC1P_MappedElement;
END_VAR
END_METHOD

METHOD SETAXISPROPERTIES
VAR_IN_OUT
	AXIS : _AXIS_REF_REAL;
	AXISPROPERTIES : L_MC1P_AxisProperties;
END_VAR
END_METHOD

METHOD UPDATEMAPPING
VAR_INPUT
	PTASKMAPLIST : POINTER TO IoStandard.IoConfigTaskMap;
	NCOUNT : DINT;
	PPDOINFOCONNECTOR : POINTER TO IoConfigConnector;
END_VAR
VAR_IN_OUT
	AXIS : _AXIS_REF_REAL;
END_VAR
END_METHOD

(* ---- L_MC1P_DRIVESPECIFIC_ENC_FREE.pou ---- *)
FUNCTION_BLOCK L_MC1P_DRIVESPECIFIC_ENC_FREE EXTENDS L_MC1P_DriveSpecific_Enc
VAR
	DRIVEINITIALIZED : BOOL;
	DRIVEINITIALIZEDERRORREASON : L_IE1P_Error;
END_VAR
END_FUNCTION_BLOCK

METHOD GETIECADRESS : BOOL
VAR_IN_OUT
	AXIS : _AXIS_REF_REAL;
	M_PPDOINFOCONNECTOR : POINTER TO IoConfigConnector;
	ATRANSELEMENT : ARRAY [1.._AXIS_REF_REAL.c_wMaxTransElem] OF L_MC1P_MappedElement;
	WTRANSELEMENTS : WORD;
	LWTRANSDATA : LWORD;
	LWRECDATA : LWORD;
	WRECEIVEELEMENTS : WORD;
	ARECEIVEELEMENT : ARRAY [1.._AXIS_REF_REAL.c_wMaxRecElem] OF L_MC1P_MappedElement;
END_VAR
END_METHOD

METHOD RECEIVEPARAMETERCALC
VAR_IN_OUT
	AXIS : _AXIS_REF_REAL;
	DATA : ARRAY [1..L_MC1P_Constants.gc_Rec_MaxDataIndex] OF POINTER TO L_MC1P_MappedElement;
END_VAR
END_METHOD

(* ---- L_MC1P_DRIVESPECIFIC_ENC_I500.pou ---- *)
FUNCTION_BLOCK L_MC1P_DRIVESPECIFIC_ENC_I500 EXTENDS L_MC1P_DriveSpecific_Enc
VAR
	PDRIVECONNECTOR : POINTER TO IoConfigConnector;
	XPOSAVAILABLE : BOOL;
	DRIVEINITIALIZED : BOOL;
	DRIVEINITIALIZEDERRORREASON : L_IE1P_Error;
END_VAR
END_FUNCTION_BLOCK

METHOD GETIECADRESS : BOOL
VAR_IN_OUT
	AXIS : _AXIS_REF_REAL;
	M_PPDOINFOCONNECTOR : POINTER TO IoConfigConnector;
	ATRANSELEMENT : ARRAY [1.._AXIS_REF_REAL.c_wMaxTransElem] OF L_MC1P_MappedElement;
	WTRANSELEMENTS : WORD;
	LWTRANSDATA : LWORD;
	LWRECDATA : LWORD;
	WRECEIVEELEMENTS : WORD;
	ARECEIVEELEMENT : ARRAY [1.._AXIS_REF_REAL.c_wMaxRecElem] OF L_MC1P_MappedElement;
END_VAR
END_METHOD

METHOD RECEIVEPARAMETERCALC
VAR_IN_OUT
	AXIS : _AXIS_REF_REAL;
	DATA : ARRAY [1..L_MC1P_Constants.gc_Rec_MaxDataIndex] OF POINTER TO L_MC1P_MappedElement;
END_VAR
END_METHOD

METHOD SETAXISPROPERTIES
VAR_IN_OUT
	AXIS : _AXIS_REF_REAL;
	AXISPROPERTIES : L_MC1P_AxisProperties;
END_VAR
END_METHOD

(* ---- L_MC1P_DRIVESPECIFIC_ENC_I950.pou ---- *)
FUNCTION_BLOCK L_MC1P_DRIVESPECIFIC_ENC_I950 EXTENDS L_MC1P_DriveSpecific_Enc
VAR_INPUT
	XCHECKCOMMUNICATIONSTATE : BOOL;
	XPOSAVAILABLE : BOOL;
END_VAR
VAR
	CIA_STATE : WORD;
	CIA_STATEOLD : WORD;
	WLENZESTATE : WORD;
	WLENZESTATE2 : WORD;
	REFCIA_STATE : REFERENCE TO WORD;
	READENCODERCRC : L_DCO_ReadDriveParameter;
	XDEVICETRANSMITTIMESVALID : BOOL;
	LRDEVICETRANSMITTIMEACTPOSMS : LREAL;
	LRDEVICETRANSMITTIMESETPOSMS : LREAL;
	PDRIVECONNECTOR : POINTER TO IoConfigConnector;
	XFDBCONFIGCHANGEDOLD : BOOL;
	XFDBCONFIGCHANGED : BOOL;
	BASICINITERROR : L_IE1P_Error;
	DRIVEINITIALIZED : BOOL;
	DRIVEINITIALIZEDERRORREASON : L_IE1P_Error;
END_VAR
END_FUNCTION_BLOCK

METHOD CHECKRESETHOMEPOS
VAR_INPUT
	WFDBSTATUSWORD : WORD;
END_VAR
VAR_IN_OUT
	AXIS : _AXIS_REF_REAL;
END_VAR
END_METHOD

METHOD DRIVECONFIGDATA
VAR_INPUT
	PCONFIGINFO : POINTER TO L_MC1P_AdditionalConfigInfo;
END_VAR
VAR_IN_OUT
	AXIS : _AXIS_REF_REAL;
END_VAR
END_METHOD

METHOD GETFDBSTATUSWORD : WORD
VAR_IN_OUT
	AXIS : _AXIS_REF_REAL;
END_VAR
END_METHOD

METHOD GETIECADRESS : BOOL
VAR_IN_OUT
	AXIS : _AXIS_REF_REAL;
	M_PPDOINFOCONNECTOR : POINTER TO IoConfigConnector;
	ATRANSELEMENT : ARRAY [1.._AXIS_REF_REAL.c_wMaxTransElem] OF L_MC1P_MappedElement;
	WTRANSELEMENTS : WORD;
	LWTRANSDATA : LWORD;
	LWRECDATA : LWORD;
	WRECEIVEELEMENTS : WORD;
	ARECEIVEELEMENT : ARRAY [1.._AXIS_REF_REAL.c_wMaxRecElem] OF L_MC1P_MappedElement;
END_VAR
END_METHOD

METHOD RECEIVEPARAMETERCALC
VAR_IN_OUT
	AXIS : _AXIS_REF_REAL;
	DATA : ARRAY [1..L_MC1P_Constants.gc_Rec_MaxDataIndex] OF POINTER TO L_MC1P_MappedElement;
END_VAR
END_METHOD

METHOD SETAXISPROPERTIES
VAR_IN_OUT
	AXIS : _AXIS_REF_REAL;
	AXISPROPERTIES : L_MC1P_AxisProperties;
END_VAR
END_METHOD

METHOD SETBASICINITIALISATION
VAR_IN_OUT
	AXIS : _AXIS_REF_REAL;
END_VAR
END_METHOD

METHOD FB_INIT : BOOL
VAR_INPUT
	BINITRETAINS : BOOL;
	BINCOPYCODE : BOOL;
END_VAR
END_METHOD

(* ---- L_MC1P_DRIVESPECIFIC_ENC_IOETC.pou ---- *)
FUNCTION_BLOCK L_MC1P_DRIVESPECIFIC_ENC_IOETC EXTENDS L_MC1P_DriveSpecific_Enc_Bpb
VAR
	CONST_ID_S131_EPM_S600 : DWORD := 16#8C13800;
	CONST_ID_S131_EPM_S601 : DWORD := 16#8C3380A;
	CONST_ID_S131_EPM_S602 : DWORD := 16#8C23801;
	CONST_ID_S131_EPM_S603 : DWORD := 16#8C4388B;
	CONST_ID_S131_EPM_S604 : DWORD := 16#9C17800;
END_VAR
END_FUNCTION_BLOCK

METHOD SETAXISPROPERTIES
VAR_IN_OUT
	AXIS : _AXIS_REF_REAL;
	AXISPROPERTIES : L_MC1P_AxisProperties;
END_VAR
END_METHOD

METHOD UPDATEMAPPING
VAR_INPUT
	PTASKMAPLIST : POINTER TO IoStandard.IoConfigTaskMap;
	NCOUNT : DINT;
	PPDOINFOCONNECTOR : POINTER TO IoConfigConnector;
END_VAR
VAR_IN_OUT
	AXIS : _AXIS_REF_REAL;
END_VAR
END_METHOD

(* ---- L_MC1P_DRIVESPECIFIC_GENERIC.pou ---- *)
FUNCTION_BLOCK L_MC1P_DRIVESPECIFIC_GENERIC EXTENDS L_MC1P_DriveSpecific_Cia402
VAR_INPUT
	ITFGENERICCONFIG : L_MC1P_IGenericAxisConfiguration;
END_VAR
END_FUNCTION_BLOCK

METHOD CALCAFTERREADINPUTS
VAR_IN_OUT
	AXIS : _AXIS_REF_REAL;
END_VAR
END_METHOD

METHOD CALCBEFOREREADINPUTS
VAR_IN_OUT
	AXIS : _AXIS_REF_REAL;
END_VAR
END_METHOD

METHOD CALCBEFOREWRITEOUTPUTS
VAR_IN_OUT
	AXIS : _AXIS_REF_REAL;
END_VAR
END_METHOD

METHOD CONTROLDRIVE : BOOL
VAR_INPUT
	XENABLE : BOOL;
END_VAR
VAR_IN_OUT
	AXIS : _AXIS_REF_REAL;
END_VAR
END_METHOD

METHOD DRIVEFAULTSTATUS : BOOL
VAR_IN_OUT
	AXIS : _AXIS_REF_REAL;
	SCSTATEINFO : L_MC1P_DriveStateCollection;
END_VAR
END_METHOD

METHOD GETADDITIONALSTATEINFOS : BOOL
VAR_IN_OUT
	AXIS : _AXIS_REF_REAL;
	SCSTATEINFO : L_MC1P_DriveStateCollection;
END_VAR
END_METHOD

METHOD HOMECONFIG : BOOL
VAR_INPUT
	LRPOSITION : LREAL;
END_VAR
VAR_OUTPUT
	WINDEX : WORD;
	BYSUBINDEX : BYTE;
	BYNROFBYTE : BYTE;
	DWDATA : DWORD;
	XWRITEPARAM : BOOL;
	XDONE : BOOL;
	XERROR : BOOL;
END_VAR
VAR_IN_OUT
	AXIS : _AXIS_REF_REAL;
	SCHOMEDATA : L_MC1P_HomeParameter;
	WSTEP : WORD;
END_VAR
END_METHOD

METHOD RECEIVEPARAMETERCALC
VAR_IN_OUT
	AXIS : _AXIS_REF_REAL;
	DATA : ARRAY [1..L_MC1P_Constants.gc_Rec_MaxDataIndex] OF POINTER TO L_MC1P_MappedElement;
END_VAR
END_METHOD

METHOD SETAXISPROPERTIES
VAR_IN_OUT
	AXIS : _AXIS_REF_REAL;
	AXISPROPERTIES : L_MC1P_AxisProperties;
END_VAR
END_METHOD

METHOD SETDRIVECONFIGINIT
VAR_IN_OUT
	AXIS : _AXIS_REF_REAL;
END_VAR
END_METHOD

METHOD TRANSMITPARAMETERCALC
VAR_IN_OUT
	AXIS : _AXIS_REF_REAL;
	DATA : ARRAY [1..L_MC1P_Constants.gc_Trans_MaxDataIndex] OF POINTER TO L_MC1P_MappedElement;
END_VAR
END_METHOD

(* ---- L_MC1P_DRIVESPECIFIC_I500.pou ---- *)
FUNCTION_BLOCK L_MC1P_DRIVESPECIFIC_I500 EXTENDS L_MC1P_DriveSpecific_CiA402
VAR_INPUT
	XFORCEACYCLICMODE : BOOL;
	WNETWORDIN1 : WORD;
	WNETWORDIN2 : WORD;
	WNETWORDIN3 : WORD;
	WNETWORDIN4 : WORD;
END_VAR
VAR_OUTPUT
	WNETWORDOUT1 : WORD;
	WNETWORDOUT2 : WORD;
END_VAR
VAR
	BRAKE : L_MC1P_BrakeControl;
	PXDUMMY : POINTER TO BOOL;
	XENABLEDRIVEOLD : BOOL;
	XDEACTIVATEPOSCTRLEXTENCERROR : BOOL;
	GETITFBRAKE : L_MC1P_IAXIS_REF_BRAKE;
END_VAR
END_FUNCTION_BLOCK

METHOD GETADDITIONALSTATEINFOS : BOOL
VAR_IN_OUT
	AXIS : _AXIS_REF_REAL;
	SCSTATEINFO : L_MC1P_DriveStateCollection;
END_VAR
END_METHOD

METHOD CHECKAVAILABLECONTROLMODE : BOOL
VAR_IN_OUT
	AXIS : _AXIS_REF_REAL;
	POSCTRLDRIVEAVAILABLE : L_IE1P_Error;
	POSCTRLPLCAVAILABLE : L_IE1P_Error;
	SPEEDCTRLDRIVEAVAILABLE : L_IE1P_Error;
	TORQUECTRLDRIVE : L_IE1P_Error;
END_VAR
END_METHOD

METHOD CONTROLDRIVE : BOOL
VAR_INPUT
	XENABLE : BOOL;
END_VAR
VAR_IN_OUT
	AXIS : _AXIS_REF_REAL;
END_VAR
END_METHOD

METHOD GETBRAKE : POINTER TO L_MC1P_BrakeControlBase
VAR_IN_OUT
	AXIS : _AXIS_REF_REAL;
END_VAR
END_METHOD

METHOD GETCAUSEOFCINH : WORD
VAR_IN_OUT
	AXIS : _AXIS_REF_REAL;
END_VAR
END_METHOD

METHOD GETIECADRESS : BOOL
VAR_IN_OUT
	AXIS : _AXIS_REF_REAL;
	M_PPDOINFOCONNECTOR : POINTER TO IoStandard.IoConfigConnector;
	ATRANSELEMENT : ARRAY [1..._AXIS_REF_REAL.c_wMaxTransElem] OF L_MC1P_MappedElement;
	WTRANSELEMENTS : WORD;
	LWTRANSDATA : LWORD;
	LWRECDATA : LWORD;
	WRECEIVEELEMENTS : WORD;
	ARECEIVEELEMENT : ARRAY [1..._AXIS_REF_REAL.c_wMaxRecElem] OF L_MC1P_MappedElement;
END_VAR
END_METHOD

METHOD GETRECEIVEDATAIMPL : DWORD
VAR_INPUT
	LWMASK : LWORD;
END_VAR
VAR_IN_OUT
	AXIS : _AXIS_REF_REAL;
END_VAR
END_METHOD

METHOD GETSTOACTIVEFROMSTATE : BOOL
VAR_IN_OUT
	AXIS : _AXIS_REF_REAL;
END_VAR
END_METHOD

METHOD GETSTATUSWORDS
VAR_OUTPUT
	STATUSWORD1 : WORD;
	STATUSWORD2 : WORD;
	STATUSWORD3 : WORD;
	STATUSWORD4 : WORD;
END_VAR
VAR_IN_OUT
	AXIS : _AXIS_REF_REAL;
END_VAR
END_METHOD

METHOD PROZESSCONTROLWORD : BOOL
VAR_IN_OUT
	AXIS : _AXIS_REF_REAL;
END_VAR
END_METHOD

METHOD RECEIVEPARAMETERCALC
VAR_IN_OUT
	AXIS : _AXIS_REF_REAL;
	DATA : ARRAY [1..L_MC1P_Constants.gc_Rec_MaxDataIndex] OF POINTER TO L_MC1P_MappedElement;
END_VAR
END_METHOD

METHOD SETAXISPROPERTIES
VAR_IN_OUT
	AXIS : _AXIS_REF_REAL;
	AXISPROPERTIES : L_MC1P_AxisProperties;
END_VAR
END_METHOD

METHOD SETAXISSTATUSWORD
VAR_IN_OUT
	AXIS : _AXIS_REF_REAL;
	DWAXISSTATUS : DWORD;
END_VAR
END_METHOD

METHOD SETBASICINITIALISATION
VAR_IN_OUT
	AXIS : _AXIS_REF_REAL;
END_VAR
END_METHOD

METHOD SETCONTROLWORDS
VAR_INPUT
	CONTROLWORD1 : WORD;
	CONTROLWORD2 : WORD;
	CONTROLWORD3 : WORD;
	CONTROLWORD4 : WORD;
END_VAR
VAR_IN_OUT
	AXIS : _AXIS_REF_REAL;
END_VAR
END_METHOD

METHOD SETDRIVECONFIGINIT
VAR_IN_OUT
	AXIS : _AXIS_REF_REAL;
END_VAR
END_METHOD

METHOD TRANSMITPARAMETERCALC
VAR_IN_OUT
	AXIS : _AXIS_REF_REAL;
	DATA : ARRAY [1..L_MC1P_Constants.gc_Trans_MaxDataIndex] OF POINTER TO L_MC1P_MappedElement;
END_VAR
END_METHOD

METHOD FB_INIT : BOOL
VAR_INPUT
	BINITRETAINS : BOOL;
	BINCOPYCODE : BOOL;
END_VAR
END_METHOD

(* ---- L_MC1P_DRIVESPECIFIC_I700.pou ---- *)
FUNCTION_BLOCK L_MC1P_DRIVESPECIFIC_I700 EXTENDS L_MC1P_DriveSpecific_CiA402
VAR_INPUT
	XSLOT2 : BOOL;
END_VAR
VAR
	ERRVALUE : L_MC1P_DriveErrValueReader;
	TPWORKER : L_MC1P_TpWorker_CiA402;
	ITFBRAKEINT : L_MC1P_IAXIS_REF_BRAKE;
	BRAKE : REFERENCE TO L_MC1P_BrakeControlBase;
	BRAKESERVICE : L_MC1P_BrakeService;
	CMDBRAKETEST : L_MC1P_AxisCommand_BrakeTest;
	CMDBRAKEGRINDIN : L_MC1P_AxisCommand_BrakeGrindIn;
	ITFCMDAUTOTUNING : L_MC1P_IAxisCommmand_Autotuning;
	WLENZECTRL : WORD;
	WLENZESTATE : WORD;
	WLENZESTATE2 : WORD;
	LRSPEEDCTRLINT : LREAL;
	LRSPEEDCTRLEXT : LREAL;
	XSETSPEEDCTRLEXT : BOOL;
	XSETSPEEDCTRLEXTOLD : BOOL;
	PSCBRAKEPAR : POINTER TO L_MC1P_BrakePara;
	PSCBRAKEPARAXIS : POINTER TO L_MC1P_BrakePara;
	PSCBRAKEGIPAR : POINTER TO L_MC1P_BrakeCmdBrakeGrindInPara;
	PSCBRAKEGIPARAXIS : POINTER TO L_MC1P_BrakeCmdBrakeGrindInPara;
	PSCBRAKETESTPAR : POINTER TO L_MC1P_BrakeCmdBrakeTestPara;
	PSCBRAKETESTPARAXIS : POINTER TO L_MC1P_BrakeCmdBrakeTestPara;
	XFDBCONFIGCHANGED : BOOL := FALSE;
	XFDBCONFIGCHANGEDOLD : BOOL := FALSE;
	READENCODERCRC : L_DCO_ReadDriveParameter;
	XIGNOREPDOINTERFACEDISABLED : BOOL;
	READQSPDRIVERAMP : L_DCO_ReadDriveParameter;
	DRIVEINITIALIZEDERRORREASON : L_IE1P_Error;
	GETITFBRAKE : L_MC1P_IAXIS_REF_BRAKE;
	GETITFCMDBRAKEGRINDIN : L_MC1P_IAxisCommmand;
	GETITFCMDBRAKETEST : L_MC1P_IAxisCommmand;
END_VAR
END_FUNCTION_BLOCK

METHOD GETADDITIONALSTATEINFOS : BOOL
VAR_IN_OUT
	AXIS : _AXIS_REF_REAL;
	SCSTATEINFO : L_MC1P_DriveStateCollection;
END_VAR
END_METHOD

METHOD GETDRIVEQSPDONE : BOOL
VAR_IN_OUT
	AXIS : _AXIS_REF_REAL;
	SCSTATEINFO : L_MC1P_DriveStateCollection;
END_VAR
END_METHOD

METHOD GETSTOACTIVEFROMSTATE : BOOL
VAR_IN_OUT
	AXIS : _AXIS_REF_REAL;
END_VAR
END_METHOD

METHOD PROZESSCONTROLWORD : BOOL
VAR_IN_OUT
	AXIS : _AXIS_REF_REAL;
END_VAR
END_METHOD

METHOD SETBRAKEITF
VAR_INPUT
	ITFBRAKE : L_MC1P_IAXIS_REF_BRAKE;
END_VAR
END_METHOD

METHOD FB_INIT : BOOL
VAR_INPUT
	BINITRETAINS : BOOL;
	BINCOPYCODE : BOOL;
END_VAR
END_METHOD

METHOD CALCAFTERREADINPUTS
VAR_IN_OUT
	AXIS : _AXIS_REF_REAL;
END_VAR
END_METHOD

METHOD CALCBEFOREWRITEOUTPUTS
VAR_IN_OUT
	AXIS : _AXIS_REF_REAL;
END_VAR
END_METHOD

METHOD CHECKRESETHOMEPOS
VAR_INPUT
	WFDBSTATUSWORD : WORD;
END_VAR
VAR_IN_OUT
	AXIS : _AXIS_REF_REAL;
END_VAR
END_METHOD

METHOD DRIVEFAULTSTATUS : BOOL
VAR_IN_OUT
	AXIS : _AXIS_REF_REAL;
	SCSTATEINFO : L_MC1P_DriveStateCollection;
END_VAR
END_METHOD

METHOD GETBRAKE : POINTER TO L_MC1P_BrakeControlBase
VAR_IN_OUT
	AXIS : _AXIS_REF_REAL;
END_VAR
END_METHOD

METHOD GETBRAKESERVICE : POINTER TO L_MC1P_BrakeService
VAR_IN_OUT
	AXIS : _AXIS_REF_REAL;
END_VAR
END_METHOD

METHOD GETCAUSEOFCINH : WORD
VAR_IN_OUT
	AXIS : _AXIS_REF_REAL;
END_VAR
END_METHOD

METHOD GETFDBSTATUSWORD : WORD
VAR_IN_OUT
	AXIS : _AXIS_REF_REAL;
END_VAR
END_METHOD

METHOD GETRECEIVEDATAIMPL : DWORD
VAR_INPUT
	LWMASK : LWORD;
END_VAR
VAR_IN_OUT
	AXIS : _AXIS_REF_REAL;
END_VAR
END_METHOD

METHOD GETSTATUSWORDS
VAR_OUTPUT
	STATUSWORD1 : WORD;
	STATUSWORD2 : WORD;
	STATUSWORD3 : WORD;
	STATUSWORD4 : WORD;
END_VAR
VAR_IN_OUT
	AXIS : _AXIS_REF_REAL;
END_VAR
END_METHOD

METHOD GETTRANSMITDATAIMPL : DWORD
VAR_INPUT
	LWMASK : LWORD;
END_VAR
VAR_IN_OUT
	AXIS : _AXIS_REF_REAL;
END_VAR
END_METHOD

METHOD GETTRANSMITDATALREALIMPL : LREAL
VAR_INPUT
	LWMASK : LWORD;
END_VAR
VAR_IN_OUT
	AXIS : _AXIS_REF_REAL;
END_VAR
END_METHOD

METHOD RECEIVEPARAMETERCALC
VAR_IN_OUT
	AXIS : _AXIS_REF_REAL;
	DATA : ARRAY [1..L_MC1P_Constants.gc_Rec_MaxDataIndex] OF POINTER TO L_MC1P_MappedElement;
END_VAR
END_METHOD

METHOD RESTOREADDITIONALRETAINDATA
VAR_INPUT
	PDATA : POINTER TO L_MC1P_uRetainData;
END_VAR
END_METHOD

METHOD SETAXISPROPERTIES
VAR_IN_OUT
	AXIS : _AXIS_REF_REAL;
	AXISPROPERTIES : L_MC1P_AxisProperties;
END_VAR
END_METHOD

METHOD SETAXISSTATUSWORD
VAR_IN_OUT
	AXIS : _AXIS_REF_REAL;
	DWAXISSTATUS : DWORD;
END_VAR
END_METHOD

METHOD SETBASICINITIALISATION
VAR_IN_OUT
	AXIS : _AXIS_REF_REAL;
END_VAR
END_METHOD

METHOD SETCONTROLWORDS
VAR_INPUT
	CONTROLWORD1 : WORD;
	CONTROLWORD2 : WORD;
	CONTROLWORD3 : WORD;
	CONTROLWORD4 : WORD;
END_VAR
VAR_IN_OUT
	AXIS : _AXIS_REF_REAL;
END_VAR
END_METHOD

METHOD SETDCBRAKE
VAR_INPUT
	XSETDCBRAKE : BOOL;
END_VAR
VAR_OUTPUT
	XDCBRAKEACTIVE : BOOL;
END_VAR
VAR_IN_OUT
	AXIS : _AXIS_REF_REAL;
END_VAR
END_METHOD

METHOD SETDRIVECONFIGINIT
VAR_IN_OUT
	AXIS : _AXIS_REF_REAL;
END_VAR
END_METHOD

METHOD SETSPEEDCTRLLIMITATION : BOOL
VAR_INPUT
	XLIMIT : BOOL;
END_VAR
VAR_IN_OUT
	AXIS : _AXIS_REF_REAL;
END_VAR
END_METHOD

METHOD SETSPEEDCTRLLOADVALUE
VAR_INPUT
	XLOAD : BOOL;
	LRVALUE : LREAL;
END_VAR
VAR_IN_OUT
	AXIS : _AXIS_REF_REAL;
END_VAR
END_METHOD

METHOD STOREADDITIONALRETAINDATA
VAR_INPUT
	PDATA : POINTER TO L_MC1P_uRetainData;
END_VAR
END_METHOD

METHOD TRANSMITPARAMETERCALC
VAR_IN_OUT
	AXIS : _AXIS_REF_REAL;
	DATA : ARRAY [1..L_MC1P_Constants.gc_Trans_MaxDataIndex] OF POINTER TO L_MC1P_MappedElement;
END_VAR
END_METHOD

(* ---- L_MC1P_DRIVESPECIFIC_I750.pou ---- *)
FUNCTION_BLOCK L_MC1P_DRIVESPECIFIC_I750 EXTENDS L_MC1P_DriveSpecific_i700
VAR
	WPPISTATE : WORD := 0;
	WPPIMODE : WORD := 0;
	WPPIACTIVATIONCYCLES : WORD := 0;
	WPPIERRORID : WORD := 0;
	WRITEPARAMETERPPI : L_DCO_WriteDriveParameter;
	WMOLSTATE : WORD := 0;
	WMOLMODE : WORD := 0;
	WMOLACTIVATIONCYCLES : WORD := 0;
	WMOLERRORID : WORD := 0;
	ITFMOLACCESS : L_MC1P_IMOLAccess;
	ITFPLIACCESS : L_MC1P_IPLIAccess;
	MOLDONE : BOOL;
	MOLERRORID : WORD;
	MOLSTATE : WORD;
	PLIACTIVE : BOOL;
	PLIERRORID : WORD;
	PLISTATE : WORD;
	PPIINVALID : BOOL;
END_VAR
END_FUNCTION_BLOCK

METHOD CALCAFTERCIA402STM : BOOL
VAR_IN_OUT
	AXIS : _AXIS_REF_REAL;
END_VAR
END_METHOD

METHOD GETADDITIONALSTATEINFOS : BOOL
VAR_IN_OUT
	AXIS : _AXIS_REF_REAL;
	SCSTATEINFO : L_MC1P_DriveStateCollection;
END_VAR
END_METHOD

METHOD GETTEXTREFIDFROMTABLE : BOOL
VAR_INPUT
	DWERRORID : DWORD;
	XSAFETYDEVICE : BOOL;
END_VAR
VAR_IN_OUT
	WTEXTREFID : WORD;
END_VAR
END_METHOD

METHOD FB_INIT : BOOL
VAR_INPUT
	BINITRETAINS : BOOL;
	BINCOPYCODE : BOOL;
END_VAR
END_METHOD

METHOD CHECKSAFETYOPTIONAVAILABLE : BOOL
VAR_INPUT
	DWPRODUCTCODE : DWORD;
END_VAR
END_METHOD

METHOD SETAXISPROPERTIES
VAR_IN_OUT
	AXIS : _AXIS_REF_REAL;
	AXISPROPERTIES : L_MC1P_AxisProperties;
END_VAR
END_METHOD

METHOD MOLSEQUENCE
VAR_IN_OUT
	AXIS : _Axis_Ref_Real;
END_VAR
END_METHOD

METHOD SETMOLSTATES
VAR_INPUT
	WSETMOLSTATE : WORD := 0;
	WSETMOLMODE : WORD := 0;
END_VAR
END_METHOD

METHOD PPISEQUENCE
VAR_IN_OUT
	AXIS : _Axis_Ref_Real;
END_VAR
END_METHOD

METHOD PPISEQUENCESTATE
END_METHOD

METHOD SETPPISTATES
VAR_INPUT
	WSETPPISTATE : WORD := 0;
	WSETPPIMODE : WORD := 0;
END_VAR
END_METHOD

(* ---- L_MC1P_DRIVESPECIFIC_I950.pou ---- *)
FUNCTION_BLOCK L_MC1P_DRIVESPECIFIC_I950 EXTENDS L_MC1P_DriveSpecific_i750
VAR
	TPWORKER2 : L_MC1P_TpWorker_CiA402;
END_VAR
END_FUNCTION_BLOCK

METHOD GETTEXTREFIDFROMTABLE : BOOL
VAR_INPUT
	DWERRORID : DWORD;
	XSAFETYDEVICE : BOOL;
END_VAR
VAR_IN_OUT
	WTEXTREFID : WORD;
END_VAR
END_METHOD

METHOD CALCAFTERREADINPUTS
VAR_IN_OUT
	AXIS : _AXIS_REF_REAL;
END_VAR
END_METHOD

METHOD CALCBEFOREWRITEOUTPUTS
VAR_IN_OUT
	AXIS : _AXIS_REF_REAL;
END_VAR
END_METHOD

METHOD CHECKSAFETYOPTIONAVAILABLE : BOOL
VAR_INPUT
	DWPRODUCTCODE : DWORD;
END_VAR
END_METHOD

METHOD GETRECEIVEDATAIMPL : DWORD
VAR_INPUT
	LWMASK : LWORD;
END_VAR
VAR_IN_OUT
	AXIS : _AXIS_REF_REAL;
END_VAR
END_METHOD

METHOD RECEIVEPARAMETERCALC
VAR_IN_OUT
	AXIS : _AXIS_REF_REAL;
	DATA : ARRAY [1..L_MC1P_Constants.gc_Rec_MaxDataIndex] OF POINTER TO L_MC1P_MappedElement;
END_VAR
END_METHOD

METHOD SETAXISPROPERTIES
VAR_IN_OUT
	AXIS : _AXIS_REF_REAL;
	AXISPROPERTIES : L_MC1P_AxisProperties;
END_VAR
END_METHOD

METHOD SETDRIVECONFIGINIT
VAR_IN_OUT
	AXIS : _AXIS_REF_REAL;
END_VAR
END_METHOD

METHOD TRANSMITPARAMETERCALC
VAR_IN_OUT
	AXIS : _AXIS_REF_REAL;
	DATA : ARRAY [1..L_MC1P_Constants.gc_Trans_MaxDataIndex] OF POINTER TO L_MC1P_MappedElement;
END_VAR
END_METHOD

(* ---- L_MC1P_DRIVESPECIFIC_I950_DRIVE.pou ---- *)
FUNCTION_BLOCK L_MC1P_DRIVESPECIFIC_I950_DRIVE EXTENDS L_MC1P_DriveSpecific_i950
VAR
	BRAKEOVERRIDE : BYTE;
	DWTARGETID : DWORD;
	XDEVICETRANSMITTIMESVALID : BOOL;
	LRDEVICETRANSMITTIMEACTPOSMS : LREAL;
	LRDEVICETRANSMITTIMESETPOSMS : LREAL;
END_VAR
END_FUNCTION_BLOCK

METHOD FB_INIT : BOOL
VAR_INPUT
	BINITRETAINS : BOOL;
	BINCOPYCODE : BOOL;
END_VAR
END_METHOD

METHOD CHECKSAFETYOPTIONAVAILABLE : BOOL
VAR_INPUT
	DWPRODUCTCODE : DWORD;
END_VAR
END_METHOD

METHOD DRIVECONFIGDATA
VAR_INPUT
	PCONFIGINFO : POINTER TO L_MC1P_AdditionalConfigInfo;
END_VAR
VAR_IN_OUT
	AXIS : _AXIS_REF_REAL;
END_VAR
END_METHOD

METHOD GETADDITIONALSTATEINFOS : BOOL
VAR_IN_OUT
	AXIS : _AXIS_REF_REAL;
	SCSTATEINFO : L_MC1P_DriveStateCollection;
END_VAR
END_METHOD

METHOD GETFDBSTATUSWORD : WORD
VAR_IN_OUT
	AXIS : _AXIS_REF_REAL;
END_VAR
END_METHOD

METHOD PROZESSCONTROLWORD : BOOL
VAR_IN_OUT
	AXIS : _AXIS_REF_REAL;
END_VAR
END_METHOD

METHOD SETAXISPROPERTIES
VAR_IN_OUT
	AXIS : _AXIS_REF_REAL;
	AXISPROPERTIES : L_MC1P_AxisProperties;
END_VAR
END_METHOD

METHOD SETAXISSTATUSWORD
VAR_IN_OUT
	AXIS : _AXIS_REF_REAL;
	DWAXISSTATUS : DWORD;
END_VAR
END_METHOD

METHOD TRANSMITPARAMETERCALC
VAR_IN_OUT
	AXIS : _AXIS_REF_REAL;
	DATA : ARRAY [1..L_MC1P_Constants.gc_Trans_MaxDataIndex] OF POINTER TO L_MC1P_MappedElement;
END_VAR
END_METHOD

(* ---- L_MC1P_DRIVESPECIFIC_I950ADV.pou ---- *)
FUNCTION_BLOCK L_MC1P_DRIVESPECIFIC_I950ADV EXTENDS L_MC1P_DriveSpecific_i950
VAR
	READDRIVEFDBCONFIG : L_DCO_ReadDriveParameter;
	READDRIVEORIENTATIONCONFIG : L_DCO_ReadDriveParameter;
	WFDBREADSTATE : WORD;
	DWLOADORIENTATIONOLD : DWORD;
	DWFEEDBACKCONFIGOLD : DWORD;
	XDRIVELOADENCODER : BOOL;
	XHOMEPOSAVAILABLEFROMAXIS : BOOL;
	XMOTORPOSAVAILABLE : BOOL;
	UACTPOSMOTORFDB : L_MC1P_PosLINT;
	DIACTPOSMOTOR : DINT;
	DIACTPOSMOTOROLD : DINT;
	DIACTVELMOTOR : DINT;
	LRACTPOSMOTORFDB : LREAL;
	LRACTVELOCITYMOTORFDB : LREAL;
END_VAR
END_FUNCTION_BLOCK

METHOD FB_INIT : BOOL
VAR_INPUT
	BINITRETAINS : BOOL;
	BINCOPYCODE : BOOL;
END_VAR
END_METHOD

METHOD PDCONVACTPOSVELMOTOR : DINT
VAR_INPUT
	DIINPUT : DINT;
END_VAR
VAR_IN_OUT
	AXIS : _AXIS_REF_REAL;
END_VAR
END_METHOD

METHOD CHECKRESETHOMEPOS
VAR_INPUT
	WFDBSTATUSWORD : WORD;
END_VAR
VAR_IN_OUT
	AXIS : _AXIS_REF_REAL;
END_VAR
END_METHOD

METHOD DRIVECONFIGDATA
VAR_INPUT
	PCONFIGINFO : POINTER TO L_MC1P_AdditionalConfigInfo;
END_VAR
VAR_IN_OUT
	AXIS : _AXIS_REF_REAL;
END_VAR
END_METHOD

METHOD GETADDITIONALSTATEINFOS : BOOL
VAR_IN_OUT
	AXIS : _AXIS_REF_REAL;
	SCSTATEINFO : L_MC1P_DriveStateCollection;
END_VAR
END_METHOD

METHOD GETFDBSTATUSWORD : WORD
VAR_IN_OUT
	AXIS : _AXIS_REF_REAL;
END_VAR
END_METHOD

METHOD GETOPTIONALACTVEL : BOOL
VAR_IN_OUT
	LRVEL : LREAL;
END_VAR
END_METHOD

METHOD HOMEPOSPERMANENTSETACTIVE : BOOL
VAR_IN_OUT
	AXIS : _AXIS_REF_REAL;
END_VAR
END_METHOD

METHOD RECEIVEPARAMETERCALC
VAR_IN_OUT
	AXIS : _AXIS_REF_REAL;
	DATA : ARRAY [1..L_MC1P_Constants.gc_Rec_MaxDataIndex] OF POINTER TO L_MC1P_MappedElement;
END_VAR
END_METHOD

METHOD SETAXISPROPERTIES
VAR_IN_OUT
	AXIS : _AXIS_REF_REAL;
	AXISPROPERTIES : L_MC1P_AxisProperties;
END_VAR
END_METHOD

(* ---- L_MC1P_ENCODERCONV.pou ---- *)
FUNCTION_BLOCK L_MC1P_ENCODERCONV
VAR_INPUT
	DIENCODERIN : DINT;
	XRESET : BOOL;
	UDIINKPERREV : UDINT := 65536;
	UDITOTALMEASURINGRANGE : UDINT := 4294967295;
	XPOSVALID : BOOL;
END_VAR
VAR_OUTPUT
	DIENCODEROUT : DINT;
	XERROR : BOOL;
	EERRORID : L_IE1P_Error;
END_VAR
VAR
	UDIENCODERSIGNAL : UDINT;
	DIENCODERINOLD : DINT;
	DIENCDIFF : DINT;
END_VAR
END_FUNCTION_BLOCK

METHOD MODULODIFF : DINT
VAR_INPUT
	DIFF : DINT;
	LEN : DWORD;
END_VAR
END_METHOD

(* ---- L_MC1P_EXTENDEDMAPPINGACCESS.pou ---- *)
FUNCTION_BLOCK L_MC1P_EXTENDEDMAPPINGACCESS
VAR
	XMAPPINGDATASUPPORT : BOOL;
	IMAPPEDINPUTCOUNT : INT;
	IMAPPEDOUTPUTCOUNT : INT;
	AMAPPEDINPUTS : ARRAY [1..maxMappedObjects] OF L_MC1P_MappedObjects;
	AMAPPEDOUTPUTS : ARRAY [1..maxMappedObjects] OF L_MC1P_MappedObjects;
	MAXMAPPEDOBJECTS : INT := 100;
END_VAR
END_FUNCTION_BLOCK

METHOD GETIECADRESS
VAR_INPUT
	AXISCONNECTOR : POINTER TO IoConfigConnector;
END_VAR
END_METHOD

METHOD GETMAPPEDDATA : POINTER TO BYTE
VAR_INPUT
	UIINDEX : WORD;
	USISUBINDEX : USINT;
	USISIZE : USINT;
	XWRITEACCESS : BOOL;
	PADDDATA : POINTER TO BYTE;
	PXWAITFORINITACCESS : POINTER TO BOOL;
END_VAR
VAR_OUTPUT
	EERRORID : L_IE1P_Error;
	XERROR : BOOL;
	USISIZEACT : USINT := 0;
END_VAR
END_METHOD

METHOD GETMAPPEDDATASUPPORT : BOOL
END_METHOD

METHOD RESETOUTPUTMAPPINGOBJECTS : BOOL
END_METHOD

METHOD SEARCHMAPPEDOBJECT : INT
VAR_INPUT
	DWNUMBER : DWORD;
	ICOUNT : INT;
	PDATA : POINTER TO L_MC1P_MappedObjects;
END_VAR
END_METHOD

(* ---- L_MC1P_EXTRA_INTERPOLATION.pou ---- *)
FUNCTION_BLOCK L_MC1P_EXTRA_INTERPOLATION
VAR_INPUT
	XENABLE : BOOL;
	LRDELAYTIME : LREAL;
	LRMAXVEL : LREAL;
	XSPEEDEQUALSZERO : BOOL;
	XTRAVERSINGRANGEMODULO : BOOL;
	XLOADPOSOFFSET : BOOL;
	LRPOSOFFSET : LREAL;
	LRCYCLELENGTH : LREAL;
	LRSETPOSIN : LREAL;
	LRSETVELIN : LREAL;
	LRSETACCIN : LREAL;
	LRSETTORQUEIN : LREAL;
	XLINEAREXTRAPOLATION : BOOL := TRUE;
END_VAR
VAR_OUTPUT
	XERROR : BOOL;
	EERRORID : L_IE1P.L_IE1P_Error;
	LRPOSOUT : LREAL;
	LRVELOUT : LREAL;
	LRACCOUT : LREAL;
	LRTORQUEOUT : LREAL;
	LRHOMINGOFFSET : LREAL;
END_VAR
VAR
	WBUFFERINDEX : WORD := 0;
	DIVALIDCOUNTER : DINT := 0;
	DISYNCTIME : DINT := 0;
	DIDELAYPRE : DINT;
	LRDELAYTIMEINT : LREAL;
	LRREMAININGTIME : LREAL;
	LRDELAYPOST : LREAL;
	LRPOSOUTSAVE : LREAL;
	LRSETPOSINOLD : LREAL;
	LRVELOUTSAVE : LREAL;
	LRACCOUTSAVE : LREAL;
	LRTORQUEOUTSAVE : LREAL;
	LRTASKCYCLE : LREAL;
	LRINVTASKCYCLE : LREAL;
	LRCYCLELENGTHINT : LREAL;
	LRRATEDVELOCITY : LREAL;
	LRHOMINGOFFSETACT : LREAL;
	ALRPOS : ARRAY [0..wBufferSize] OF LREAL;
	ALRPOSROUNDS : ARRAY [0..wBufferSize] OF LREAL;
	ALRVEL : ARRAY [0..wBufferSize] OF LREAL;
	ALRACC : ARRAY [0..wBufferSize] OF LREAL;
	ALRTORQUE : ARRAY [0..wBufferSize] OF LREAL;
	LRVELOUTOLD : LREAL;
	LRPOSOUTOLD : LREAL;
	XENABLEOLD : BOOL;
	XENABLED : BOOL;
	XSPEEDEQUALSZEROINT : BOOL;
	XTRAVERSINGRANGEMODULOINT : BOOL;
	LRPOSOUTTEMP1 : LREAL;
	LRPOSOUTTEMP2 : LREAL;
	XPARAMETERSCHANGED : BOOL;
	XLOADPOSOFFSETOLD : BOOL;
	XOLDPOSINVALID : BOOL;
	WBUFFERSIZE : WORD := 31;
END_VAR
END_FUNCTION_BLOCK

METHOD CALCFILTERVALUES
END_METHOD

METHOD DETECTOVERFLOW
VAR_INPUT
	LRACTPOS : LREAL;
	LRPOSOLD : LREAL;
	LRACTCOUNTER : LREAL;
END_VAR
VAR_OUTPUT
	LRNEWCOUNTER : LREAL;
END_VAR
END_METHOD

METHOD ENABLEINIT
END_METHOD

METHOD EXTRAPOLATION
END_METHOD

METHOD GETVELOCITY : LREAL
END_METHOD

METHOD INITBUFFER
END_METHOD

METHOD INTERPOLATION
END_METHOD

METHOD LOADOFFSET
VAR_INPUT
	OFFSET : LREAL;
END_VAR
END_METHOD

METHOD READINPUTDATA
END_METHOD

METHOD RESETOUTPUTS
END_METHOD

(* ---- L_MC1P_FASTOUTPUT.pou ---- *)
FUNCTION_BLOCK L_MC1P_FASTOUTPUT EXTENDS L_MC1P_Template
VAR_INPUT
	XEXECUTE : BOOL;
	XABORT : BOOL;
	BYDIGITALOUTPUTSEL : BYTE := 1;
	XOUTPUTSTATE : BOOL;
	LRSWITCHPOSITION : LREAL;
	WEXTERNALDELAYCOMPENSATION : WORD;
	LRDYNVELPOSOFFSET : LREAL;
	XRESET : BOOL;
	XDISABLEACCCALC : BOOL := FALSE;
	EVALUESOURCE : MC_SOURCE := MC_SOURCE.mcActualValue;
END_VAR
VAR_OUTPUT
	XDONE : BOOL;
	XBUSY : BOOL;
	XCOMMANDABORTED : BOOL;
	XERROR : BOOL;
	EERRORID : L_IE1P_Error;
END_VAR
VAR_IN_OUT
	FASTIO_OUT : L_FastIO_OutRef;
END_VAR
VAR
	BEXCECUTEOLD : BOOL;
	BABORTEDOLD : BOOL;
	BRESETOLD : BOOL;
	FOUTPUTTIMERTICK : LREAL;
	BEXECUTEEDGE : BOOL;
	FPOSDIFF : LREAL;
	FLASTPOSDIFF : LREAL;
	SNPOSDIFFCALCCOUNTER : SINT;
	RES : INT;
	WRINGBUFFERINDEX : WORD;
	LRVELRINGBUFFER : ARRAY [0..wEncFilterCycles] OF LREAL;
	LRVELFILTERBUFFERSUM : LREAL;
	LRPOSDIFFINFILT : LREAL;
	XFLAGBUFFERFULL : BOOL;
	LRAXISPOSITION : LREAL;
	LRAXISVELOCITY : LREAL;
	LRAXISACCELERATION : LREAL;
	FOUTPUTTIMERTICKTRIGGEREVENT : LREAL;
	LRDELAYCOMPENSATION : LREAL := 0;
	XDONTSWITCH : BOOL;
	XBUSYINTERN : BOOL := FALSE;
	BYDIGITALOUTPUTSEL_INT : BYTE := 1;
	XOUTPUTSTATE_INT : BOOL;
	LRSWITCHPOSITION_INT : LREAL;
	WEXTERNALDELAYCOMPENSATION_INT : WORD;
	LRDYNVELPOSOFFSET_INT : LREAL;
	XDISABLEACCCALC_INT : BOOL := FALSE;
	EVALUESOURCE_INT : MC_SOURCE;
	BYMAXOUTPCOUNT : BYTE;
	LRDELAYFACTOR : LREAL;
	PENCFREETMP : POINTER TO _AXIS_REF_ENC;
	EENCTYPE : L_Mc1P_EncoderType;
	WENCFILTERCYCLES : WORD := 10;
END_VAR
END_FUNCTION_BLOCK

METHOD CALCULATESWITCHTIME : LREAL
VAR_IN_OUT
	AXIS : AXIS_REF;
END_VAR
END_METHOD

METHOD CHECKSWITCHPOSITIONOVERRUN : BOOL
VAR_IN_OUT
	AXIS : AXIS_REF;
END_VAR
END_METHOD

METHOD FREEZEINPUTS
END_METHOD

METHOD GETTIMERTICKFORATONCEOUTPUTSETTING : LREAL
VAR_IN_OUT
	AXIS : AXIS_REF;
END_VAR
END_METHOD

METHOD INSERTENTRYINTOFIFO : INT
VAR_INPUT
	LRTIMERTICK : LREAL;
	BSTATE : BOOL;
END_VAR
VAR_IN_OUT
	AXIS : AXIS_REF;
	FASTIO_OUT : L_FastIO_OutRef;
END_VAR
END_METHOD

METHOD RESETALLFBOUTPUTS
END_METHOD

(* ---- L_MC1P_FINISHPOSITIONING.pou ---- *)
FUNCTION_BLOCK L_MC1P_FINISHPOSITIONING EXTENDS L_MC1P_Template
VAR_INPUT
	XENABLE : BOOL;
	XFINISHPOSITIONING : BOOL;
	XMOVELASTSETPOS : BOOL;
	XCONTINUOUSUPDATE : BOOL;
	LRVELOCITY : LREAL;
	LRACCELERATION : LREAL;
	LRDECELERATION : LREAL;
	LRJERK : LREAL;
END_VAR
VAR_OUTPUT
	XVALID : BOOL;
	XACTIVE : BOOL;
	XDONE : BOOL;
	XCOMMANDABORTED : BOOL;
	XERROR : BOOL;
	EERRORID : L_IE1P_Error;
	XTARGETPOSVALID : BOOL;
	LRLASTTARGETPOS : LREAL;
	LRDISTANCETARGETPOS : LREAL;
	LRLASTSETPOS : LREAL;
	LRDISTANCELASTSETPOS : LREAL;
END_VAR
VAR
	FB_FP : L_MC1P_FinishPositioning_internal;
END_VAR
END_FUNCTION_BLOCK

(* ---- L_MC1P_FINISHPOSITIONING_INTERNAL.pou ---- *)
FUNCTION_BLOCK L_MC1P_FINISHPOSITIONING_INTERNAL EXTENDS L_MC1P_Template_IntFB
VAR_INPUT
	XENABLE : BOOL;
	XFINISHPOSITIONING : BOOL;
	XMOVELASTSETPOS : BOOL;
	XCONTINUOUSUPDATE : BOOL;
	LRVELOCITY : LREAL;
	LRACCELERATION : LREAL;
	LRDECELERATION : LREAL;
	LRJERK : LREAL;
END_VAR
VAR_OUTPUT
	XVALID : BOOL;
	XACTIVE : BOOL;
	XDONE : BOOL;
	XCOMMANDABORTED : BOOL;
	XERROR : BOOL;
	EERRORID : L_IE1P_Error;
	XTARGETPOSVALID : BOOL;
	LRLASTTARGETPOS : LREAL;
	LRDISTANCETARGETPOS : LREAL;
	LRLASTSETPOS : LREAL;
	LRDISTANCELASTSETPOS : LREAL;
END_VAR
VAR
	LRTARGETPOS_INT : LREAL;
	XEXECUTE_INT : BOOL;
	EDIRECTION_INT : MC_DIRECTION;
	XFINISHPOSITIONINGOLD : BOOL;
	XMOVELASTSETPOSOLD : BOOL;
	FBMB : L_MC1P_MoveBasic := STRUCT(wCalcProfileMode := 1);
	XBUSY_INT : BOOL;
	XCALCULATE : BOOL;
	XENABLEOLD : BOOL;
	XUSED : BOOL;
END_VAR
END_FUNCTION_BLOCK

METHOD MAIN
VAR_IN_OUT
	AXIS : AXIS_REF;
	FBBASE : L_MC1P_Template_ForAxis;
END_VAR
END_METHOD

(* ---- L_MC1P_FOLLOWSETVALUES.pou ---- *)
FUNCTION_BLOCK L_MC1P_FOLLOWSETVALUES EXTENDS L_MC1P_Template_Licence_150
VAR_INPUT
	XEXECUTE : BOOL;
	XCONTINUOUSUPDATE : BOOL;
	LRPOSITION : LREAL;
	LRVELOCITY : LREAL;
	LRACCELERATION : LREAL;
	ESETVALUEMODE : L_MC1P_SetValueMode := L_MC1P_SetValueMode.Pos;
END_VAR
VAR_OUTPUT
	XBUSY : BOOL;
	XCOMMANDABORTED : BOOL;
	XERROR : BOOL;
	EERRORID : L_IE1P_Error;
END_VAR
VAR
	FSV : L_MC1P_FollowSetValues_internal;
	USESPEEDCTRLMODE : BOOL;
END_VAR
END_FUNCTION_BLOCK

(* ---- L_MC1P_FOLLOWSETVALUES_INTERNAL.pou ---- *)
FUNCTION_BLOCK L_MC1P_FOLLOWSETVALUES_INTERNAL EXTENDS L_MC1P_Template_Edge
VAR_INPUT
	XCONTINUOUSUPDATE : BOOL := TRUE;
	LRPOSITION : LREAL;
	LRVELOCITY : LREAL := 0;
	LRACCELERATION : LREAL := 0;
	ESETVALUEMODE : L_MC1P_SetValueMode;
END_VAR
VAR
	XCONTINUOUSUPDATEINT : BOOL;
	EWARNINGID : L_IE1P_Error;
	EWARNINGIDOLD : L_IE1P_Error;
	XSLSWARNINGACTIVE : BOOL;
	XPOSPROFILERINUSE : BOOL;
	PG_INT : REFERENCE TO L_MC1P_PosProfiler;
	PG_LIMITER : L_MC1P_PosProfilerClutchState;
	RG : L_MC1P_RampGeneratorIntern;
	XFOLLOWERPOSMODE : BOOL;
	XRESETSLSPOSOFFSET : BOOL;
	XPOSPROFILERCLUTCHACTIVE : BOOL;
	XPOSPROFILERCLUTCHACTIVEOLD : BOOL;
	LRPOSDISTSLSRESET : LREAL;
	LRINTEGRATORAPPPOS : LREAL;
	LRINTEGRATORPOSSLS : LREAL;
	LRFOLLOWINGERRORSLS : LREAL;
	XPG_LIMITERDONEOLD : BOOL;
	LRSETPOSITIONAPP : LREAL;
	LRSETPOSITIONAPPOLD : LREAL;
	LRSETVELOCITYAPP : LREAL;
	LRSETVELOCITYAPPOLD : LREAL;
	LRSETACCELERATIONAPP : LREAL := 0.0;
	LRSETSLAVEPOS : LREAL;
	LRSETSLAVEVEL : LREAL;
	LRSETSLAVEACC : LREAL;
	XSLSACTIVEOLD : BOOL;
	LRSLSDECELERATIONOLD : LREAL;
	XIGNOREACCFORPOSINTEGRATION : BOOL;
	XUSESPEEDCTRLMODE : BOOL;
	LRSETACCDECOLD : LREAL;
	LRSLSDECELERATION : LREAL;
	FUNCTIONTYPE : L_MC1P_TypeFunction;
	IGNOREACCFORPOSINTEGRATION : BOOL;
	POSPROFILERINUSE : BOOL;
	USESPEEDCTRLMODE : BOOL;
END_VAR
END_FUNCTION_BLOCK

METHOD ABORT
VAR_IN_OUT
	AXIS : AXIS_REF;
	FBBASE : L_MC1P_Template;
END_VAR
END_METHOD

METHOD CYCLIC
VAR_IN_OUT
	AXIS : AXIS_REF;
	FBBASE : L_MC1P_Template;
END_VAR
END_METHOD

METHOD INIT
VAR_IN_OUT
	AXIS : AXIS_REF;
	FBBASE : L_MC1P_Template;
END_VAR
END_METHOD

METHOD PROCESSFOLLOWERSLS
VAR_INPUT
	LRSETVEL : LREAL;
	LRSETACC : LREAL;
END_VAR
VAR_OUTPUT
	LRSETSLSPOSLIMIT : LREAL;
	LRSETSLSVELLIMIT : LREAL;
	LRSETSLSACCLIMIT : LREAL;
END_VAR
VAR_IN_OUT
	AXIS : AXIS_REF;
END_VAR
END_METHOD

METHOD RESETSLSFOLLOWINGERROR
VAR_OUTPUT
	LRSETSLSPOSLIMIT : LREAL;
	LRSETSLSVELLIMIT : LREAL;
	LRSETSLSACCLIMIT : LREAL;
END_VAR
VAR_IN_OUT
	AXIS : AXIS_REF;
END_VAR
END_METHOD

(* ---- L_MC1P_FORCESETVALUES.pou ---- *)
FUNCTION_BLOCK L_MC1P_FORCESETVALUES EXTENDS L_MC1P_SetSetValueManipulator
VAR_INPUT
	LRFORCEDPOSITION : LREAL;
	LRFORCEDVELOCITY : LREAL;
	LRFORCEDACCELERATION : LREAL;
	LRFORCEDTORQUE : LREAL;
END_VAR
END_FUNCTION_BLOCK

METHOD CALCULATE2
VAR_IN_OUT
	AXIS : Axis_REf;
END_VAR
END_METHOD

(* ---- L_MC1P_FREEENCODERSIMULATION.pou ---- *)
FUNCTION_BLOCK L_MC1P_FREEENCODERSIMULATION
VAR_INPUT
	POSITIONSOURCE : L_MC1P_IAXIS_REF_POOL;
	ENCODERAXIS : L_MC1P_IEncoderInterface;
	XUSEACTVALUES : BOOL := TRUE;
	WDELAY : WORD := 1;
	LRNOISEAMP : LREAL := 0.0;
	DWNOISESEEDVALUETOSET : DWORD := 0;
	XENABLENOISE : BOOL := TRUE;
	LRRESOLUTION : LREAL := 0.0;
	LROFFSET : LREAL;
	LRSLIPPINGFACTOR : LREAL := 0;
	ALRHARMONICPERIOD : ARRAY [1..wMaxHarmonics] OF LREAL;
	ALRHARMONICPHASE : ARRAY [1..wMaxHarmonics] OF LREAL;
	ALRHARMONICAMPLITUDE : ARRAY [1..wMaxHarmonics] OF LREAL;
	LRHARMONICCYCLELENGTH : LREAL;
	LRENCCYCLETIME : LREAL := -1;
	XFORCEERROR : BOOL;
	DIFORCEDENCODERSIGNAL : DINT := 0;
END_VAR
VAR_OUTPUT
	DWNOISESEEDVALUEACT : DWORD;
END_VAR
VAR
	PAXISREF : POINTER TO AXIS_REF;
	NOISE : L_UMTP_RandomGenerator;
	WNOISEMODE : WORD := 0;
	LRPOSIN : LREAL;
	LRENCODERPOS : LREAL;
	LRENCODERPOSOLD : LREAL;
	UDIENCODERPOS : UDINT;
	ADELAYBUFFER : ARRAY [1..wBufferSize] OF LREAL;
	WWRITEIDX : WORD;
	WREADIDX : WORD := 1;
	WREADIDXOLD : WORD := 1;
	DIROUNDSIN : DINT;
	LRPOSINOLD : LREAL;
	LRACTTIME : LREAL;
	LRNEXTUPDATETIME : LREAL;
	IDX : WORD;
	LRSLIPPINGOFFSET : LREAL;
	PAXISREAL : POINTER TO _AXIS_REF_REAL;
	LRHARMONICERROR : LREAL;
	PPBYTE : POINTER TO POINTER TO BYTE;
	PBADRESSCIASTATEINIT : POINTER TO BYTE;
	PBADRESSLENZESTATE2INIT : POINTER TO BYTE;
	PBPOSADRESSINIT : POINTER TO BYTE;
	PBMICSECTICKSINIT : POINTER TO BYTE;
	PBABSCOUNTERINIT : POINTER TO BYTE;
	DIENCODERPOSITIONINITIAL : DINT;
	CIA_STATE : WORD := 16#64;
	LENZESTATE2 : WORD := 16#C00;
	WENCODERTYPE : WORD;
	PENCAXIS : POINTER TO _AXIS_REF_ENC;
	_DIENCODERPOSITION : DINT;
	_UDIMEASURINGRANGE : UDINT;
	XAXISSIMULATIONACTIVE : BOOL;
	PUDIDUMMY : POINTER TO UDINT;
	XOPERATIONAL : BOOL;
	LWRECDATA : LWORD;
	_WMICSECTICKS : WORD;
	PDIENCODERPOS : POINTER TO DINT := ADR(_diEncoderPosition);
	PWMICSECTICKS : POINTER TO WORD := ADR(_wMicSecTicks);
	_DWMICSECTICKS : DWORD;
	PDWABSCOUNTER : POINTER TO DWORD := ADR(_dwMiCSecTicks);
	DWTIMESTAMP : DWORD;
	WBUFFERSIZE : WORD := 50;
	WMAXDELAY : WORD := (wBufferSize - 1);
	WMAXHARMONICS : WORD := 5;
	COMMSIMULATION : L_MC1P_ICommmunicationSimulation;
	GETRECIEVEDATACONFIG : LWORD;
	GETTRANSMITDATACONFIG : LWORD;
	LOADFDB : LREAL;
	RECIEVEELEMCOUNT : WORD;
	RECIEVEELEMENT : POINTER TO L_MC1P_MappedElement;
	RECIEVEELEMENTADRESS : POINTER TO ARRAY [1..L_MC1P_Constants.gc_Rec_MaxDataIndex] OF POINTER TO L_MC1P_MappedElement;
	TRANSELEMCOUNT : WORD;
	TRANSELEMENT : POINTER TO L_MC1P_MappedElement;
	TRANSELEMENTADRESS : POINTER TO ARRAY [1..L_MC1P_Constants.gc_Trans_MaxDataIndex] OF POINTER TO L_MC1P_MappedElement;
END_VAR
END_FUNCTION_BLOCK

METHOD GETENCODERTYPE : WORD
VAR_INPUT
	PAXIS : POINTER TO _Axis_ref_real;
END_VAR
END_METHOD

METHOD GETMEASURINGRANGE : UDINT
END_METHOD

METHOD ACTIVATESIMULATION
VAR_IN_OUT
	AXIS : _AXIS_REF_REAL;
END_VAR
END_METHOD

METHOD CALCULATEINPUTDATA
VAR_IN_OUT
	AXIS : _AXIS_REF_REAL;
END_VAR
END_METHOD

METHOD CALCULATEOUTPUTDATA
VAR_IN_OUT
	AXIS : _AXIS_REF_REAL;
END_VAR
END_METHOD

METHOD DISABLESIMULATION
VAR_IN_OUT
	AXIS : _AXIS_REF_REAL;
END_VAR
END_METHOD

METHOD GETCOMMSTATE : L_DCO.L_DCO_CommState
VAR_INPUT
	PAXISCOMM : POINTER TO _AXIS_REF_COM;
END_VAR
END_METHOD

METHOD GETSDOERROR : WORD
VAR_INPUT
	DWERRORCODE : DWORD;
END_VAR
END_METHOD

METHOD PARREAD
VAR_INPUT
	WIDX : DWORD;
END_VAR
END_METHOD

METHOD PARREAD_GETOUTPUT
VAR_INPUT
	WIDX : DWORD;
END_VAR
VAR_OUTPUT
	SZDATAREAD : CAA_SIZE;
	XDONE : BOOL;
	XERROR : BOOL;
	WERROR : WORD;
END_VAR
END_METHOD

METHOD PARREAD_SETINPUT
VAR_INPUT
	WIDX : DWORD;
	XEXECUTE : BOOL;
	WINDEX : WORD;
	BYSUBINDEX : BYTE;
	PBUFFER : POINTER TO BYTE;
	SZSIZE : UDINT;
	UDITIMEOUT : UDINT;
	XSLOTB : BOOL;
END_VAR
END_METHOD

METHOD PARWRITE
VAR_INPUT
	WIDX : DWORD;
END_VAR
END_METHOD

METHOD PARWRITE_GETOUTPUT
VAR_INPUT
	WIDX : DWORD;
END_VAR
VAR_OUTPUT
	XDONE : BOOL;
	XERROR : BOOL;
	WERROR : WORD;
END_VAR
END_METHOD

METHOD PARWRITE_SETINPUT
VAR_INPUT
	WIDX : DWORD;
	XEXECUTE : BOOL;
	WINDEX : WORD;
	BYSUBINDEX : BYTE;
	PBUFFER : POINTER TO BYTE;
	SZSIZE : UDINT;
	UDITIMEOUT : UDINT;
	XSLOTB : BOOL;
END_VAR
END_METHOD

METHOD RESTARTMASTER
VAR_INPUT
	XEXECUTE : BOOL;
	PAXIS : POINTER TO _AXIS_REF_COM;
END_VAR
VAR_OUTPUT
	XDONE : BOOL;
	XERROR : BOOL;
	XBUSY : BOOL;
	DWERROR : DWORD;
END_VAR
END_METHOD

(* ---- L_MC1P_GEARBOXPOSITIONBASE.pou ---- *)
FUNCTION_BLOCK L_MC1P_GEARBOXPOSITIONBASE
VAR_INPUT
	XENABLE : BOOL;
	LRPOSX : LREAL;
	DWNUMERATOR : DWORD := 1;
	DWDENOMINATOR : DWORD := 1;
	XLOADPOSY : BOOL;
	LRLOADPOSY : LREAL;
	LNLOADPOSYRESIDUAL : LINT;
END_VAR
VAR_OUTPUT
	LRPOSY : LREAL;
	LNACTPOSYRESIDUAL : LINT;
	XERROR : BOOL := FALSE;
	EERRORID : L_IE1P_Error := 0;
END_VAR
VAR
	XINIT : BOOL := FALSE;
	LNPOSX : LINT := 0;
	LNPOSY : LINT := 0;
	LNPOSXOLD : LINT := 0;
	LNPOSXDIFF : LINT := 0;
	LNPOSYDIFF : LINT := 0;
	LNPOSYOLD : LINT := 0;
	LNRES_GEARBOX : LINT := 0;
	LRLENX : LREAL;
	LRLENY : LREAL;
	LRLENXOLD : LREAL;
	LRLENYOLD : LREAL;
END_VAR
END_FUNCTION_BLOCK

METHOD CALL_S000_CYCLIC
END_METHOD

METHOD CALL_ERRORHANDLER
END_METHOD

METHOD CALL_RESET
END_METHOD

METHOD L_HLPMODULOADD : LREAL
VAR_INPUT
	LRINPUT : LINT;
	LROFFSET : LINT;
	LRLENGHT : LINT;
END_VAR
END_METHOD

METHOD L_HLPMODULODIFF : LREAL
VAR_INPUT
	LRDIFF : LINT;
	LRLEN : LINT;
END_VAR
END_METHOD

METHOD L_HLPMULDIV : LREAL
VAR_INPUT
	LNINPUT : LINT;
	DWNUMERATOR : DWORD;
	DWDENOMINATOR : DWORD;
	PLNRES : POINTER TO LINT;
END_VAR
END_METHOD

(* ---- L_MC1P_GENERICAXISCONFIGURATION.pou ---- *)
FUNCTION_BLOCK L_MC1P_GENERICAXISCONFIGURATION
VAR_INPUT
	WSCALEREVTOINCMODE : WORD := 1;
	LRINCPERREV : LREAL := 10000;
	WSCALEUNITTOSPEEDMODE : WORD := 1;
	LRSCALEUNITTOSPEEDFACTOR : LREAL := 1;
	XDIFFERENTSPEEDTOUNITFACTOR : BOOL;
	LRSCALESPEEDTOUNITFACTOR : LREAL := 1;
	XREFTORQUESUPPORTED : BOOL;
	LRREFTORQUEUNITFACTOR : LREAL := 0.001;
	LRDEFAULTMOTORTORQUE : LREAL := 1;
	DITORQUEREFVALUE : DINT := 1000;
END_VAR
VAR
	DRIVEHOMINGSUPPORTED : BOOL;
	FBINSTANCE : POINTER TO L_MC1P_GenericAxisConfiguration;
	RETAINMODE : WORD;
END_VAR
END_FUNCTION_BLOCK

METHOD CALCAFTERREADINPUTS
VAR_IN_OUT
	AXIS : _AXIS_REF_REAL;
	DRIVESPECIFIC : L_MC1P_DriveSpecific_Generic;
END_VAR
END_METHOD

METHOD CALCBEFOREREADINPUTS
VAR_IN_OUT
	AXIS : _AXIS_REF_REAL;
	DRIVESPECIFIC : L_MC1P_DriveSpecific_Generic;
END_VAR
END_METHOD

METHOD CALCBEFOREWRITEOUTPUTS
VAR_IN_OUT
	AXIS : _AXIS_REF_REAL;
	DRIVESPECIFIC : L_MC1P_DriveSpecific_Generic;
END_VAR
END_METHOD

METHOD DRIVECONFIG
VAR_INPUT
	WOFFSET : WORD;
END_VAR
VAR_OUTPUT
	XCONFIGBUSY : BOOL;
	XWAITFORPARAMETERWRITEDONE : BOOL;
	XWAITFORPARAMETERREADDONE : BOOL;
	XREADSTRING : BOOL;
	DWWRITEDATA : DWORD;
	WINDEX : WORD;
	BYSUBINDEX : BYTE;
	BYNROFBYTE : BYTE;
END_VAR
VAR_IN_OUT
	AXIS : _AXIS_REF_REAL;
	CONFIGINFO : L_MC1P_AdditionalConfigInfo;
	WSTEP : WORD;
	EERRORID : WORD;
	DWREADDATA : DWORD;
	SREADDATA : STRING(255);
END_VAR
END_METHOD

METHOD GETADDITIONALSTATEINFOS : BOOL
VAR_IN_OUT
	AXIS : _AXIS_REF_REAL;
	DRIVESPECIFIC : L_MC1P_DriveSpecific_Generic;
	SCSTATEINFO : L_MC1P_DriveStateCollection;
END_VAR
END_METHOD

METHOD GETHOMINGSTATE
VAR_INPUT
	WHOMESTATE : WORD;
END_VAR
VAR_IN_OUT
	AXIS : _AXIS_REF_REAL;
	XHOMEPOSAVAILABLEDRIVE : BOOL;
END_VAR
END_METHOD

METHOD HOMECONFIG
VAR_INPUT
	LRPOSITION : LREAL;
END_VAR
VAR_OUTPUT
	XCONFIGBUSY : BOOL;
	XERROR : BOOL;
	WINDEX : WORD;
	BYSUBINDEX : BYTE;
	BYNROFBYTE : BYTE;
	DWDATA : DWORD;
	XWRITEPARAM : BOOL;
END_VAR
VAR_IN_OUT
	AXIS : _AXIS_REF_REAL;
	SCHOMEDATA : L_MC1P_HomeParameter;
	WSTEP : WORD;
END_VAR
END_METHOD

METHOD RECEIVEPARAMETERCALC
VAR_IN_OUT
	AXIS : _AXIS_REF_REAL;
	DATA : ARRAY [1...L_MC1P_Constants.gc_Rec_MaxDataIndex] OF POINTER TO L_MC1P_MappedElement;
	DRIVESPECIFIC : L_MC1P_DriveSpecific_Generic;
END_VAR
END_METHOD

METHOD TRANSMITPARAMETERCALC
VAR_IN_OUT
	AXIS : _AXIS_REF_REAL;
	DATA : ARRAY [1...L_MC1P_Constants.gc_Trans_MaxDataIndex] OF POINTER TO L_MC1P_MappedElement;
	DRIVESPECIFIC : L_MC1P_DriveSpecific_Generic;
END_VAR
END_METHOD

(* ---- L_MC1P_GETDIRECTION.pou ---- *)
FUNCTION_BLOCK L_MC1P_GETDIRECTION
VAR_INPUT
	LRCYCSETPOSIN : LREAL;
	LRCYCSETVELIN : LREAL;
	ETRAVERSINGRANGE : L_MC1P_TraversingRange;
	LRCYCLELENGTH : LREAL;
END_VAR
VAR_OUTPUT
	XPOSITIVE : BOOL := FALSE;
	XNEGATIVE : BOOL := FALSE;
	XSTANDSTILL : BOOL := TRUE;
	EACTDIRECTION : MC_DIRECTION := MC_DIRECTION.mcCurrentDirection;
END_VAR
VAR
	LRPOSDIFF : LREAL;
	ALRPOSDIFF : ARRAY [1..10] OF LREAL := [0, 0, 0, 0, 0, 0, 0, 0, 0, 0];
	BYCOUNTER : BYTE := 1;
	LRCYCSETPOSIN_OLD : LREAL;
	I : BYTE := 1;
	LRSUMMEPOSDIFF : LREAL;
	XFIRSTCYCLESTANDSTILL : BOOL := TRUE;
	LRPOSITIONSTANDSTILL : LREAL;
	LRTHRESHOLDPOS : LREAL;
	LRTHRESHOLDNEG : LREAL;
	XPOSITIVEDRIFT : BOOL;
	XNEGATIVEDRIFT : BOOL;
	LRMIN : LREAL;
	LRMAX : LREAL;
	LRHYST : LREAL;
	XHYSTFOUND : BOOL;
	LRVARIANCE : LREAL := 1E-06;
	LRTMPMIN : LREAL;
	LRTMPMAX : LREAL;
	ICOUNT : INT;
	XINITDONE : BOOL := FALSE;
	LRMITTELWERT_ENCODER : LREAL;
	XOPERATIONENABLEDOLD : BOOL;
	LRVELDIFF : LREAL;
	LRFACTOR : LREAL := 500;
	LRFACTOR_INT : LREAL;
	XENCODERCHANGE : BOOL := FALSE;
	LRMITTELWERT : LREAL := 0;
	XOPERATIONENABLED : BOOL;
	LRTASKCYCLE : LREAL;
	LRSETEXTERNALTHRESHOLD_INT : LREAL;
	LRREFOFFSETACTINT : LREAL;
	XINAXISREF : BOOL;
	WAXISINITSTATE : WORD;
	WAXISINITSTATEOLD : WORD;
	XAXISOPERATIONENABLED : BOOL;
	XINITTASKCYCLE : BOOL := TRUE;
	WAXISMODE : WORD;
	CLRVARIANCE : LREAL := 1E-09;
END_VAR
END_FUNCTION_BLOCK

METHOD ISBETWEEN : BOOL
VAR_INPUT
	LRVALUE : LREAL;
	LRUPPER : LREAL;
	LRLOWER : LREAL;
	LRVARIANCE : LREAL := 1E-09;
END_VAR
END_METHOD

METHOD ISOUTSIDE : BOOL
VAR_INPUT
	LRVALUE : LREAL;
	LRUPPER : LREAL;
	LRLOWER : LREAL;
	LRVARIANCE : LREAL := 1E-09;
END_VAR
END_METHOD

METHOD RESETVLAUES
END_METHOD

METHOD SETAXISVALUES
VAR_INPUT
	WMODE : WORD;
	WINITSTATE : WORD;
	XOPERATIONENABLED : BOOL;
END_VAR
END_METHOD

METHOD SETEXTERNALTHRESHOLD : LREAL
VAR_INPUT
	LRSETEXTERNALTHRESHOLD : LREAL;
END_VAR
END_METHOD

METHOD SETREFOFFSETACT
VAR_INPUT
	LRREFOFFSETACT : LREAL;
END_VAR
END_METHOD

(* ---- L_MC1P_GETMAXVELACCDEC.pou ---- *)
FUNCTION_BLOCK L_MC1P_GETMAXVELACCDEC EXTENDS L_MC1P_Template
VAR_INPUT
	XENABLE : BOOL;
	DWTIMESTAMP : DWORD;
	EMC_SOURCE : MC_SOURCE;
END_VAR
VAR_OUTPUT
	XVALID : BOOL;
	XBUSY : BOOL;
	XERROR : BOOL;
	EERRORID : L_IE1P_Error;
	LRMAXVELOCITIY : LREAL;
	DWTIMEVELATMAX : DWORD;
	LRMAXACCELERATION : LREAL;
	DWTIMEACCATMAX : DWORD;
	LRMAXDECELERATION : LREAL;
	DWTIMEDECATMAX : DWORD;
END_VAR
VAR
	XENABLEOLD : BOOL := FALSE;
	EMC_SOURCEOLD : MC_SOURCE;
	XINITDONE : BOOL := FALSE;
	LRACCELERATION : LREAL;
	LRDECELERATION : LREAL;
	LRVELOCITIY : LREAL;
END_VAR
END_FUNCTION_BLOCK

METHOD FB_RESET : BOOL
END_METHOD

(* ---- L_MC1P_GETTPVALUE.pou ---- *)
FUNCTION_BLOCK L_MC1P_GETTPVALUE
VAR_INPUT
	XENABLE : BOOL;
	TPRECDATA : L_MC1P_TpReceiveData;
	LRVALUE : LREAL;
	LRTIMEDELAY : LREAL;
	LRCYCLELENGTH : LREAL;
END_VAR
VAR_OUTPUT
	XBUSY : BOOL;
	XERROR : BOOL;
	EERRORID : L_IE1P_Error;
	XTPRECEIVED : BOOL;
	LRTPVALUE : LREAL;
END_VAR
VAR
	ALRRINGBUFFER : ARRAY [0..(wRingBufferDepth - 1)] OF LREAL;
	XINITDONE : BOOL;
	WINITCYCLES : WORD;
	DITIMESTAMPDIFF : DINT;
	LRTASKCYCLE_NS : LREAL;
	LRTASKCYCLETIME : LREAL;
	DWTIMESTAMPOLD : DWORD;
	WVALUEIDX : WORD;
	LRINTERVAL : LREAL;
	UDIINTERVAL : UDINT;
	LRFACTOR : LREAL;
	LRBASE : LREAL;
	LRDIFF : LREAL;
	DIVALUEBASE : DINT;
	DWTMP : DWORD;
	LRTMP : LREAL;
	WRINGBUFFERDEPTH : WORD := 21;
END_VAR
END_FUNCTION_BLOCK

METHOD CALL_RINGBUFFER
END_METHOD

METHOD FB_INIT : BOOL
VAR_INPUT
	BINITRETAINS : BOOL;
	BINCOPYCODE : BOOL;
END_VAR
END_METHOD

(* ---- L_MC1P_HALT_INTERNAL.pou ---- *)
FUNCTION_BLOCK L_MC1P_HALT_INTERNAL EXTENDS L_MC1P_Template_IntFB
VAR_INPUT
	EXECUTE : BOOL;
	DECELERATION : LREAL;
	JERK : LREAL;
	BUFFERMODE : MC_BUFFER_MODE;
	CALLEDBYABC : BOOL;
	CONTINUOUSUPDATE : BOOL;
END_VAR
VAR_OUTPUT
	DONE : BOOL;
	BUSY : BOOL;
	ACTIVE : BOOL;
	COMMANDABORTED : BOOL;
	ERROR : BOOL;
	ERRORID : L_IE1P_Error;
END_VAR
VAR
	FBMB : L_MC1P_MoveBasic := STRUCT(wCalcProfileMode := 1);
	XUSED : BOOL;
END_VAR
END_FUNCTION_BLOCK

METHOD MAIN
VAR_IN_OUT
	AXIS : AXIS_REF;
	FBBASE : L_MC1P_Template_ForAxis;
END_VAR
END_METHOD

METHOD RESET
VAR_IN_OUT
	FBBASE : L_MC1P_Template_ForAxis;
END_VAR
END_METHOD

(* ---- L_MC1P_HLPRAMPGENERATOR.pou ---- *)
FUNCTION_BLOCK L_MC1P_HLPRAMPGENERATOR
VAR_INPUT
	LRACC : LREAL := 0;
	LRDEC : LREAL := 0;
	LRVEL : LREAL := 0;
	LRJERKACC : LREAL := 0;
	LRJERKDEC : LREAL := 0;
	LRTASKCYCLE : LREAL := 0;
	XRESET : BOOL := FALSE;
	XACCDECHISTORY : BOOL := FALSE;
END_VAR
VAR_OUTPUT
	LRSETPOS : LREAL := 0;
	LRSETVEL : LREAL := 0;
	LRSETACCDEC : LREAL := 0;
	DNSTATE : DINT := 0;
END_VAR
VAR
	C_RG_ACC : WORD := 0;
	C_RG_DEC : WORD := 1;
	C_RG_MINJERK : LREAL := 0;
	C_RG_STATE_INI : DINT := 0;
	C_RG_STATE_CNS : DINT := 1;
	C_RG_STATE_ACC : DINT := 2;
	C_RG_STATE_DEC : DINT := 3;
	ALRACCLIMIT : ARRAY [0..1] OF LREAL;
	ALRJERKABS : ARRAY [0..1] OF LREAL;
	LRVELINTERNAL : LREAL;
	DWINDEX : DWORD;
	LRVELDIFF : LREAL;
	LRVELCOMPARE : LREAL;
	LRACCINTERNAL : LREAL;
	LRTEMP : LREAL;
	VELCOMPMAX : LREAL;
	VELCOMPMIN : LREAL;
	INDEX_TEMP : DINT;
END_VAR
END_FUNCTION_BLOCK

METHOD CALCDELTAVEL
END_METHOD

METHOD CALCJERK : LREAL
VAR_INPUT
	VEL : LREAL;
	ACC : LREAL;
END_VAR
END_METHOD

METHOD SETSTARTVALUESINTERN
VAR_INPUT
	LRVEL : LREAL := 0;
	LRACC : LREAL := 0;
	LRTASKCYCLE : LREAL := 0;
END_VAR
END_METHOD

METHOD SETSTARTVALUES
VAR_INPUT
	LRVEL : LREAL := 0;
	LRACC : LREAL := 0;
END_VAR
END_METHOD

(* ---- L_MC1P_HOME_INTERNAL.pou ---- *)
FUNCTION_BLOCK L_MC1P_HOME_INTERNAL EXTENDS L_MC1P_Template_IntFB
VAR_INPUT
	EXECUTE : BOOL;
	POSITION : LREAL;
	BUFFERMODE : MC_BUFFER_MODE;
	HOMEABSSWITCH : BOOL;
	USEEXTPARAMETER : BOOL;
	EXTPARAMETER : L_MC1P_HomeParameter;
	EXTTP : MC_TRIGGER_REF;
END_VAR
VAR_OUTPUT
	DONE : BOOL;
	BUSY : BOOL;
	ACTIVE : BOOL;
	COMMANDABORTED : BOOL;
	ERROR : BOOL;
	ERRORID : L_IE1P_Error;
END_VAR
VAR
	XEXECUTEOLD : BOOL;
	XRESETOUTPUT : BOOL;
	EACTSTATE : L_MC1P_AXIS_STATE;
	WFUNID : WORD;
	AWSEQTYPE : ARRAY [1..c_MaxSeqCount] OF WORD;
	AWSEQMASK : ARRAY [1..c_MaxSeqCount] OF WORD;
	AXSEQPARA2 : ARRAY [1..c_MaxSeqCount] OF BOOL;
	AXSEQDIRCCW : ARRAY [1..c_MaxSeqCount] OF BOOL;
	AXSEQTORQUELIM : ARRAY [1..c_MaxSeqCount] OF BOOL;
	AWSEQJMPMASK : ARRAY [1..c_MaxSeqCount] OF WORD;
	AWSEQJMPCNT : ARRAY [1..c_MaxSeqCount] OF WORD;
	AXPREPARETP : ARRAY [1..c_MaxSeqCount] OF BOOL;
	XTPMODE : BOOL;
	XPARASET2 : BOOL;
	WSTEP : WORD;
	WSEQCNT : WORD;
	WSEQCNTTMP : WORD;
	WSEQTYPE : WORD;
	XINTENABLETRAJECTORY : BOOL;
	PG : REFERENCE TO L_MC1P_PosProfiler;
	SCHOMEPROFILE : L_MC1P_ProfileParameter;
	LRACTIVEHOMEPOSITION : LREAL;
	DWSIGNALSTATE : DWORD;
	XDIRCCW : BOOL;
	XINTMARKERABORT : BOOL;
	XINTMARKEREXECUTE : BOOL;
	XINTSTOPBYABORT : BOOL;
	LRTRQLIMTIMER : LREAL;
	SCHOMEPARAMETER : L_MC1P_HomeParameter;
	SCTP : MC_TRIGGER_REF;
	GETTP : L_MC1P_TouchProbe_Internal;
	ABORTTP : L_MC1P_AbortTrigger_Internal;
	L_DCO_WRITEDRIVEPARAMETER1 : L_DCO_WriteDriveParameter;
	PXDUMMY : POINTER TO BOOL;
	XBUFFERACTIVE : BOOL;
	XTRIGGERACTIVE : BOOL;
	XDONEOLD : BOOL;
	LRACTTORQUELIMIT : LREAL;
	DWINSTANCE : __XWORD;
	PAXIS : POINTER TO _AXIS_REF_REAL;
	WRINGBUFFERINDEX : WORD;
	LRVELRINGBUFFER : ARRAY [0..L_MC1P_Constants.gc_EncFilterCyclesMax] OF LREAL;
	LRVELFILTERBUFFERSUM : LREAL;
	LRACTVELFILTER : LREAL;
	WENCFILTERCYCLES : WORD := 10;
	WIGNORE : WORD;
	TIMETPDETECT : DWORD;
	XIGNORETP : BOOL;
	XINTMARKERABORTACTIVE : BOOL;
	XINTMARKEREXECUTEACTIVE : BOOL;
	SCPROFILEDATATMP : L_MC1P_ProfileData;
	SCHOMEPROFILETMP : L_MC1P_ProfileParameter;
	SCHOMEPROFILELIM : L_MC1P_ProfileParameter;
	XLIMITOLD : BOOL;
	XPOSSWLIMIT : BOOL;
	XNEGSWLIMIT : BOOL;
	XWARNING : BOOL;
	XWARNINGOLD : BOOL;
	EWARNINGID : L_IE1P_Error;
	EWARNINGIDOLD : L_IE1P_Error;
	XLOGINFO : BOOL;
	ELOGINFOID : L_IE1P_Error;
	ELOGINFOIDOLD : L_IE1P_Error;
	XUSED : BOOL;
	XCALLFROMAXESGROUP : BOOL := FALSE;
	ETMPHOMEMODE : L_MC1P_HomeMode;
	LRTMPOFFSETPOSITION : LREAL;
	XPOSPROFILERINUSE : BOOL;
	C_DEFAULT : WORD := 2#0;
	C_HWLIMPOS : WORD := 2#1;
	C_NOTHWLIMPOS : WORD := 2#10;
	C_HWLIMNEG : WORD := 2#100;
	C_NOTHWLIMNEG : WORD := 2#1000;
	C_REFMARKPOS : WORD := 2#10000;
	C_REFMARKNEG : WORD := 2#100000;
	C_TPDETECTED : WORD := 2#1000000;
	C_TORQUELIMDELAY : WORD := 2#10000000;
	C_MAXSEQCOUNT : WORD := 8;
	POSPROFILERINUSE : BOOL;
END_VAR
END_FUNCTION_BLOCK

METHOD ABORTHOMING
VAR_IN_OUT
	AXIS : AXIS_REF;
	FBBASE : L_MC1P_Template_ForAxis;
END_VAR
END_METHOD

METHOD HOMECONTROLERBASED
VAR_IN_OUT
	AXIS : AXIS_REF;
	FBBASE : L_MC1P_Template_ForAxis;
END_VAR
END_METHOD

METHOD HOMEDRIVEBASED
VAR_IN_OUT
	AXIS : AXIS_REF;
	FBBASE : L_MC1P_Template_ForAxis;
END_VAR
END_METHOD

METHOD MAIN
VAR_IN_OUT
	AXIS : AXIS_REF;
	FBBASE : L_MC1P_Template_ForAxis;
END_VAR
END_METHOD

METHOD RESETHOMING
VAR_IN_OUT
	AXIS : AXIS_REF;
	FBBASE : L_MC1P_Template_ForAxis;
END_VAR
END_METHOD

METHOD SETCALLFROMAXESGROUP
VAR_INPUT
	XSETCALLFROMAXESGROUP : BOOL;
END_VAR
END_METHOD

METHOD CALLHOMEFUNCTIONS
VAR_IN_OUT
	AXIS : AXIS_REF;
	FBBASE : L_MC1P_Template_ForAxis;
END_VAR
END_METHOD

METHOD CHECKHOMEPARAMETER : BOOL
VAR_IN_OUT
	AXIS : AXIS_REF;
END_VAR
END_METHOD

METHOD CHECKPOWERDIRECTION : BOOL
VAR_IN_OUT
	AXIS : AXIS_REF;
END_VAR
END_METHOD

METHOD DELETEPREPARETPSIGNAL
END_METHOD

METHOD GETCAPTUREVALUE : LREAL
END_METHOD

METHOD HOMEDGEMANAGER
END_METHOD

METHOD HOMGENERATESIGNALS
VAR_IN_OUT
	AXIS : AXIS_REF;
END_VAR
END_METHOD

METHOD HOMGETPARAMETERS
VAR_IN_OUT
	AXIS : AXIS_REF;
	FBBASE : L_MC1P_Template_ForAxis;
END_VAR
END_METHOD

METHOD HOMLIMITER
VAR_IN_OUT
	AXIS : AXIS_REF;
	FBBASE : L_MC1P_Template_ForAxis;
END_VAR
END_METHOD

METHOD HOMPROFILEABORT
END_METHOD

METHOD HOMPROFILEEXECUTE
END_METHOD

METHOD SEQUENCEABORT
VAR_IN_OUT
	AXIS : AXIS_REF;
	FBBASE : L_MC1P_Template_ForAxis;
END_VAR
END_METHOD

METHOD SEQUENCEDEFAULT
VAR_IN_OUT
	AXIS : AXIS_REF;
END_VAR
END_METHOD

METHOD SEQUENCEGOAGAIN
VAR_IN_OUT
	AXIS : AXIS_REF;
	FBBASE : L_MC1P_Template_ForAxis;
END_VAR
END_METHOD

METHOD SEQUENCEMOVESETREF
VAR_IN_OUT
	AXIS : AXIS_REF;
	FBBASE : L_MC1P_Template_ForAxis;
END_VAR
END_METHOD

METHOD SEQUENCEPOSITIONING
VAR_IN_OUT
	AXIS : AXIS_REF;
	FBBASE : L_MC1P_Template_ForAxis;
END_VAR
END_METHOD

METHOD SEQUENCETESTSIGNAL
VAR_IN_OUT
	AXIS : AXIS_REF;
END_VAR
END_METHOD

METHOD SETSEQUENCE
VAR_INPUT
	WSEQEL : WORD;
	WSEQTYPE : WORD;
	WSEQMASK : WORD;
	XSEQPARA2 : BOOL;
	XSEQDIRCCW : BOOL;
	XSEQTORQUELIM : BOOL;
	WSEQJMPMASK : WORD;
	WSEQJMPCNT : WORD;
	XPREPARETP : BOOL := FALSE;
END_VAR
END_METHOD

(* ---- L_MC1P_HWLIMITSWITCHINTERFACE.pou ---- *)
FUNCTION_BLOCK L_MC1P_HWLIMITSWITCHINTERFACE EXTENDS L_MC1P_Template
VAR_INPUT
	XENABLE : BOOL;
	XLIMITSWITCHPOS : BOOL;
	XLIMITSWITCHNEG : BOOL;
	XOVERWRITEOTHERSOURCES : BOOL;
END_VAR
VAR_OUTPUT
	XBUSY : BOOL;
	XERROR : BOOL;
	EERRORID : L_IE1P_Error;
END_VAR
VAR
	PXDUMMY : POINTER TO BOOL;
	PWDUMMY : POINTER TO WORD;
	XENABLEOLD : BOOL;
END_VAR
END_FUNCTION_BLOCK

(* ---- L_MC1P_IECVARACCESSOEM_BASE.pou ---- *)
FUNCTION_BLOCK L_MC1P_IECVARACCESSOEM_BASE
VAR
	_VARACCESSIBASE : IBase;
	_PPIVARACCESS4 : POINTER TO IecVarAccessLibrary.IIecVarAccess4;
	_VARACCESS4 : IecVarAccessLibrary.IIecVarAccess4;
	_PPIVARACCESS5 : POINTER TO IecVarAccessLibrary.IIecVarAccess5;
	_VARACCESS5 : IecVarAccessLibrary.IIecVarAccess5;
	_VARINFO : VariableInformationStruct;
END_VAR
END_FUNCTION_BLOCK

METHOD FB_EXIT : BOOL
VAR_INPUT
	BINCOPYCODE : BOOL;
END_VAR
END_METHOD

METHOD FB_INIT
VAR_INPUT
	BINITRETAINS : BOOL;
	BINCOPYCODE : BOOL;
END_VAR
END_METHOD

METHOD OPENIECVARACCESS : BOOL
END_METHOD

(* ---- L_MC1P_IECVARACCESSOEM_SYMBOL.pou ---- *)
FUNCTION_BLOCK L_MC1P_IECVARACCESSOEM_SYMBOL EXTENDS L_MC1P_IecVarAccessOEM_Base
VAR
	_HNODE : ICollections.IBaseTreeNode;
END_VAR
END_FUNCTION_BLOCK

METHOD FINDSYMBOL : SysTypes.RTS_IEC_RESULT
VAR_INPUT
	PNODE : ICollections.IBaseTreeNode;
	DWADDRESS : DWORD;
END_VAR
VAR_IN_OUT
	SVARIABLENAMESPACE : STRING(255);
END_VAR
END_METHOD

METHOD FINDSYMBOL_ : SysTypes.RTS_IEC_RESULT
VAR_INPUT
	PNODE : ICollections.IBaseTreeNode;
	DWADDRESS : DWORD;
END_VAR
VAR_IN_OUT
	SVARIABLENAMESPACE : STRING(255);
END_VAR
END_METHOD

METHOD GETADDRESS : __XWORD
VAR_OUTPUT
	RESULT : SysTypes.RTS_IEC_RESULT;
END_VAR
END_METHOD

METHOD GETSYMBOL : SysTypes.RTS_IEC_RESULT
VAR_INPUT
	DWADDRESS : DWORD;
END_VAR
VAR_IN_OUT
	SVARIABLENAMESPACE : STRING(255);
END_VAR
END_METHOD

METHOD INITIALIZE : BOOL
VAR_INPUT
	SVARIABLENAMESPACE : STRING(255);
END_VAR
END_METHOD

(* ---- L_MC1P_INTEGRATEAXIS.pou ---- *)
FUNCTION_BLOCK L_MC1P_INTEGRATEAXIS
VAR_INPUT
	LRCYCVEL : LREAL;
	XLOADSTARTPOS : BOOL;
	LRSTARTPOS : LREAL;
	LRCYCLELENGTH : LREAL;
END_VAR
VAR_OUTPUT
	LRSETPOSOUT : LREAL;
	LRSETVELOUT : LREAL;
	XERROR : BOOL;
	EERRORID : L_IE1P_Error;
END_VAR
VAR
	LRLENGTH : LREAL;
	LRSPEED : LREAL;
	LRPOS : LREAL;
	LRDIFF : LREAL;
	LRDIFF2 : LREAL;
	LRTASKCYCLE : LREAL;
END_VAR
END_FUNCTION_BLOCK

(* ---- L_MC1P_LIMITER.pou ---- *)
FUNCTION_BLOCK L_MC1P_LIMITER EXTENDS L_MC1P_Template
VAR_INPUT
	XENABLE : BOOL;
	DWLIMITERCONTROL : DWORD;
END_VAR
VAR_OUTPUT
	XBUSY : BOOL;
	XERROR : BOOL;
	EERRORID : L_IE1P_Error;
	DWSTATE : DWORD;
	XLIMITATIONACTIVE : BOOL;
	XSLSACTIVE : BOOL;
	LRACTLIMITEDVELOCITY : LREAL;
	LRACTLIMITEDDECTIME : LREAL;
	LRACTLIMITEDJERK : LREAL;
END_VAR
VAR
	PXDUMMY : POINTER TO BOOL;
	PDWDUMMY : POINTER TO DWORD;
	XSLSCHANGES : BOOL;
	XSLSNEWACTIVEDECELERATION : BOOL;
	XLIMITATIONSLSACTIVE : BOOL;
	XLIMITATIONDIRECTIONACTIVE : BOOL;
	XSAFESTOPACTIVE : BOOL;
	XENABLEOLD : BOOL;
	XRESETOUTPUT : BOOL;
	DWCONTROL_INT : DWORD;
	DWLIMITERCONTROL_INT : DWORD;
	PWDUMMY : POINTER TO WORD;
END_VAR
END_FUNCTION_BLOCK

(* ---- L_MC1P_MANIPULATIONBASE.pou ---- *)
FUNCTION_BLOCK L_MC1P_MANIPULATIONBASE EXTENDS L_MC1P_Template
VAR_INPUT
	XENABLE : BOOL;
	EEXECUTIONINDEX : L_MC1P_ExecutionIndex := L_MC1P_ExecutionIndex.First;
END_VAR
VAR_OUTPUT
	XBUSY : BOOL;
	XACTIVE : BOOL;
	XERROR : BOOL;
	EERRORID : L_IE1P.L_IE1P_Error;
	LRSETPOSOUT : LREAL;
	LRSETVELOUT : LREAL;
	LRSETACCOUT : LREAL;
	LRSETTORQUEOUT : LREAL;
END_VAR
VAR
	XENABLEOLD : BOOL;
	XFUNENABLEOLD : BOOL;
	XFUNRESETOLD : BOOL;
	XLOADPOSOFFSETOLD : BOOL;
	XWAITFORDISABLED : BOOL;
	EEXECUTIONINDEXINT : WORD;
	XERRORWRITEITF : BOOL;
	XERRORREADINPUTS : BOOL;
	LRSETPOSIN : LREAL;
	LRSETVELIN : LREAL;
	LRSETACCIN : LREAL;
	LRSETTORQUEIN : LREAL;
	LRPOSOUT : LREAL;
	LRVELOUT : LREAL;
	LRACCOUT : LREAL;
	LRTORQUEOUT : LREAL;
	XFIRSTSTANDSTILL : BOOL;
	XFIRSTSTANDSTILLOLD : BOOL;
	LRSETPOSOUTOLD : LREAL;
	XNUMERICALCORRACCIN : BOOL := TRUE;
	ACCELERATIONCORRECTION : BOOL;
END_VAR
END_FUNCTION_BLOCK

METHOD CALLCYCLIC2
VAR_IN_OUT
	AXIS : Axis_REf;
END_VAR
END_METHOD

METHOD CONNECTTOAXIS
VAR_IN_OUT
	AXIS : Axis_Ref;
END_VAR
END_METHOD

METHOD DISCONNECTFROMAXIS
VAR_IN_OUT
	AXIS : Axis_Ref;
END_VAR
END_METHOD

METHOD READINPUTS2
VAR_IN_OUT
	AXIS : Axis_REf;
END_VAR
END_METHOD

METHOD RESETOUTPUTS2
VAR_IN_OUT
	AXIS : Axis_REf;
END_VAR
END_METHOD

METHOD CALCULATE2
VAR_IN_OUT
	AXIS : Axis_REf;
END_VAR
END_METHOD

METHOD CHECKINPUTDATA2
VAR_IN_OUT
	AXIS : Axis_REf;
END_VAR
END_METHOD

METHOD ENABLEEXIT2
VAR_IN_OUT
	AXIS : Axis_REf;
END_VAR
END_METHOD

METHOD ENABLEINIT2
VAR_IN_OUT
	AXIS : Axis_REf;
END_VAR
END_METHOD

METHOD LOADOFFSET2
VAR_INPUT
	OFFSET : LREAL;
END_VAR
VAR_IN_OUT
	AXIS : Axis_REf;
END_VAR
END_METHOD

METHOD RESET2
VAR_IN_OUT
	AXIS : Axis_REf;
END_VAR
END_METHOD

METHOD CALCVALUES
VAR_INPUT
	XENABLE : BOOL;
	XRESET : BOOL;
	LRSETPOS : LREAL;
	LRSETVEL : LREAL;
	LRSETACC : LREAL;
	LRSETTORQUE : LREAL;
	XLOADPOSOFFSET : BOOL;
	LRPOSOFFSET : LREAL;
END_VAR
VAR_OUTPUT
	XACTIVE : BOOL;
	XERROR : BOOL;
	EERRORID : L_IE1P.L_IE1P_Error;
	LRSETPOSOUT : LREAL;
	LRSETVELOUT : LREAL;
	LRSETACCOUT : LREAL;
	LRSETTORQUEOUT : LREAL;
END_VAR
VAR_IN_OUT
	AXIS : Axis_REf;
END_VAR
END_METHOD

METHOD FILTERSTARTCONDITION
VAR_INPUT
	LRSETPOS : LREAL;
	LRSETVEL : LREAL;
	LRSETACC : LREAL;
END_VAR
VAR_IN_OUT
	AXIS : Axis_ref;
END_VAR
END_METHOD

(* ---- L_MC1P_MANJOGOPENLOOP.pou ---- *)
FUNCTION_BLOCK L_MC1P_MANJOGOPENLOOP EXTENDS L_MC1P_Template
VAR_INPUT
	XENABLE : BOOL;
	XJOGPOSITIVE : BOOL;
	XJOGNEGATIVE : BOOL;
	XPARAMETERSET2 : BOOL;
END_VAR
VAR_OUTPUT
	XBUSY : BOOL;
	XOPERATIONENABLED : BOOL;
	XDONE : BOOL;
	XACTIVE : BOOL;
	XCOMMANDABORTED : BOOL;
	XERROR : BOOL;
	EERRORID : L_IE1P_Error;
END_VAR
VAR
	WFUNID : WORD;
	XENABLEOLD : BOOL;
	PAXISREAL : POINTER TO _AXIS_REF_REAL;
	XREGULATORON : BOOL := FALSE;
	XPOWSTATUS : BOOL := FALSE;
	XPOWVALID : BOOL := FALSE;
	WFBID : WORD := 0;
	ITFMOLACCESS : L_MC1P_IMOLAccess;
	WMOLSTATE : WORD := 0;
	WMOLMODE : WORD := 0;
	WJOGSTATE : WORD := 0;
	WJOGSTATEOLD : WORD := 0;
	LRCYCLECOUNT : LREAL := 0;
	XINITNEGATIVE : BOOL := 0;
	XJOGSTATEOLD : BOOL := 0;
	XDISABLING : BOOL := FALSE;
	XABORTALLOWED : BOOL;
	XDIRECTIONALLOWED : BOOL;
	EALLOWEDSERVICEDIRECTION : L_MC1P_ServiceDirection := L_MC1P_ServiceDirection.both;
END_VAR
END_FUNCTION_BLOCK

(* ---- L_MC1P_MANUALJOG.pou ---- *)
FUNCTION_BLOCK L_MC1P_MANUALJOG EXTENDS L_MC1P_Template_Licence_150
VAR_INPUT
	XJOGPOSITIVE : BOOL;
	XJOGNEGATIVE : BOOL;
	XCONTINUOUSUPDATE : BOOL;
	LRVELOCITY : LREAL;
	LRACCELERATION : LREAL;
	LRDECELERATION : LREAL;
	LRJERK : LREAL;
	XSTEPMODE : BOOL;
	LRDISTANCE : LREAL;
END_VAR
VAR_OUTPUT
	XDONE : BOOL;
	XBUSY : BOOL;
	XCOMMANDABORTED : BOOL;
	XERROR : BOOL;
	EERRORID : L_IE1P_Error;
END_VAR
VAR
	MANJOG : L_MC1P_ManualJog_Internal;
END_VAR
END_FUNCTION_BLOCK

(* ---- L_MC1P_MANUALJOG_INTERNAL.pou ---- *)
FUNCTION_BLOCK L_MC1P_MANUALJOG_INTERNAL EXTENDS L_MC1P_Template_IntFB
VAR_INPUT
	XJOGPOSITIVE : BOOL;
	XJOGNEGATIVE : BOOL;
	XCONTINUOUSUPDATE : BOOL;
	LRVELOCITY : LREAL;
	LRACCELERATION : LREAL;
	LRDECELERATION : LREAL;
	LRJERK : LREAL;
	LRJERKDEC : LREAL;
	XSTEPMODE : BOOL;
	LRDISTANCE : LREAL;
END_VAR
VAR_OUTPUT
	XBUSY : BOOL;
	XDONE : BOOL;
	XCOMMANDABORTED : BOOL;
	XERROR : BOOL;
	EERRORID : L_IE1P_Error;
END_VAR
VAR
	FBSTOP : L_MC1P_Halt_Internal;
	FBMOVEVELOCITY : L_MC1P_MoveVelocity_Internal;
	FBMOVERELATIVE : L_MC1P_MoveRelative_Internal;
	PGMOVEVEL : L_MC1P_PosProfilerOptDecUsage;
	PGMOVEREL : L_MC1P_PosProfilerOptDecUsage;
	STATE : INT;
	XJOGPOSITIVEOLD : BOOL;
	XJOGNEGATIVEOLD : BOOL;
	XERRORINTOLD : BOOL;
	XERRORINT : BOOL;
	EERRORIDINT : L_IE1P_Error;
	XSTOPBYERROR : BOOL;
	XMASTERINSTANCE : BOOL;
	LRVELOCITY_INT : LREAL;
	LRACCELERATION_INT : LREAL;
	LRDECELERATION_INT : LREAL;
	LRJERK_INT : LREAL;
	LRJERKDEC_INT : LREAL;
	PXDUMMY : POINTER TO BOOL;
	XHALTFIRSTCYCLE : BOOL;
	XUSED : BOOL;
	XSTEPMODE_INT : BOOL;
	XSTEPMODEOLD_INT : BOOL;
	LRDISTANCE_INT : LREAL;
	XSLIACTIVEOLD : BOOL;
	XSTOPBYSTEPMODE : BOOL;
	XSTOPBYSTEPMODEDONE : BOOL;
	ABORTEDBYLIMIT : BOOL;
END_VAR
END_FUNCTION_BLOCK

METHOD HALT
VAR_IN_OUT
	AXIS : AXIS_REF;
	FBBASE : L_MC1P_Template_ForAxis;
END_VAR
END_METHOD

METHOD JOGNEG
VAR_IN_OUT
	AXIS : AXIS_REF;
	FBBASE : L_MC1P_Template_ForAxis;
END_VAR
END_METHOD

METHOD JOGPOS
VAR_IN_OUT
	AXIS : AXIS_REF;
	FBBASE : L_MC1P_Template_ForAxis;
END_VAR
END_METHOD

METHOD MAIN
VAR_IN_OUT
	AXIS : AXIS_REF;
	FBBASE : L_MC1P_Template_ForAxis;
END_VAR
END_METHOD

METHOD RESETINOUT
END_METHOD

METHOD SETSTOPBYERROR : BOOL
END_METHOD

(* ---- L_MC1P_MEANENCODERPOSITIONFILTER.pou ---- *)
FUNCTION_BLOCK L_MC1P_MEANENCODERPOSITIONFILTER EXTENDS L_UBUP_MemoryProvider
VAR_INPUT
	WENCFILTERCYCLES : WORD;
	LRTASKCYCLE : LREAL;
END_VAR
VAR
	FILTER : L_USPP_AverageFilterRecursive;
	DIENCODERPOSIN : DINT;
	ALRRINGBUFFER : ARRAY [0..c_wEncFilterCyclesMax] OF LREAL;
	LRFILTERTIMEROLD : LREAL;
	LRTASKCYCLEINT : LREAL;
	WFILTERSTATE : WORD;
	C_WENCFILTERCYCLESMAX : WORD := 300;
	PTR : POINTER TO BYTE;
	SIZE : UDINT;
END_VAR
END_FUNCTION_BLOCK

METHOD FB_INIT : BOOL
VAR_INPUT
	BINITRETAINS : BOOL;
	BINCOPYCODE : BOOL;
END_VAR
END_METHOD

METHOD CALCULATE
VAR_INPUT
	LRCYCPOSIN : LREAL;
	LRCYCVELIN : LREAL;
END_VAR
VAR_OUTPUT
	LRCYCPOSOUT : LREAL;
	LRCYCVELOUT : LREAL;
	WFILTERSTATE : WORD;
END_VAR
END_METHOD

METHOD INIT
END_METHOD

METHOD RESET
END_METHOD

(* ---- L_MC1P_MEANVALUEFILTER.pou ---- *)
FUNCTION_BLOCK L_MC1P_MEANVALUEFILTER
VAR_INPUT
	WFILTERCYCLES : WORD := 1;
	DIINPUT : DINT;
	XRESET : BOOL;
END_VAR
VAR_OUTPUT
	DIOUTPUT : DINT;
END_VAR
VAR
	XRESETOLD : BOOL;
	WFILTERCYCLESINT : WORD;
	WFILTERCYCLESOLD : WORD;
	WRINGBUFFERINDEX : WORD;
	LIFILTERBUFFERSUM : LINT;
	ADIRINGBUFFER : ARRAY [0..c_wEncFilterCyclesMax] OF DINT;
	C_WENCFILTERCYCLESMAX : WORD := 100;
END_VAR
END_FUNCTION_BLOCK

(* ---- L_MC1P_MEANVALUEFILTERPOS.pou ---- *)
FUNCTION_BLOCK L_MC1P_MEANVALUEFILTERPOS
VAR_INPUT
	WFILTERCYCLES : WORD;
	DIPOSIN : DINT;
	XRESET : BOOL;
END_VAR
VAR_OUTPUT
	DIPOSOUT : DINT;
	LRRESIDUAL : LREAL;
END_VAR
VAR
	XRESETOLD : BOOL;
	WFILTERCYCLESINT : WORD;
	WFILTERCYCLESOLD : WORD;
	WRINGBUFFERINDEX : WORD;
	LIFILTERBUFFERSUM : LINT;
	ADIRINGBUFFER : ARRAY [0..c_wEncFilterCyclesMax] OF DINT;
	DICORRECTCYCLES : DINT := 0;
	C_WENCFILTERCYCLESMAX : WORD := 100;
END_VAR
END_FUNCTION_BLOCK

(* ---- L_MC1P_MEANVALUEFILTERPOSLREAL.pou ---- *)
FUNCTION_BLOCK L_MC1P_MEANVALUEFILTERPOSLREAL
VAR_INPUT
	WFILTERCYCLES : WORD;
	LRPOSIN : LREAL;
	XRESET : BOOL;
END_VAR
VAR_OUTPUT
	LRPOSOUT : LREAL;
END_VAR
VAR
	XRESETOLD : BOOL;
	WFILTERCYCLESINT : WORD;
	WFILTERCYCLESOLD : WORD;
	WRINGBUFFERINDEX : WORD;
	LRFILTERBUFFERSUM : LREAL;
	ALRRINGBUFFER : ARRAY [0..c_wEncFilterCyclesMax] OF LREAL;
	C_WENCFILTERCYCLESMAX : WORD := 100;
END_VAR
END_FUNCTION_BLOCK

(* ---- L_MC1P_MEASUREDISTANCE.pou ---- *)
FUNCTION_BLOCK L_MC1P_MEASUREDISTANCE EXTENDS L_MC1P_Template
VAR_INPUT
	XENABLE : BOOL;
	EMC_SOURCE : MC_SOURCE;
END_VAR
VAR_OUTPUT
	XVALID : BOOL;
	XBUSY : BOOL;
	XERROR : BOOL;
	EERRORID : L_IE1P_Error;
	LRDISTANCE : LREAL;
END_VAR
VAR
	EMC_SOURCE_INT : MC_SOURCE;
	XENABLEOLD : BOOL := FALSE;
	XINITDONE : BOOL := FALSE;
	LRSTARTPOS : LREAL;
	LRPOSNEW : LREAL;
	LRPOSOLD : LREAL;
	LRROUNDS : LREAL;
	LRDIFF : LREAL;
END_VAR
END_FUNCTION_BLOCK

METHOD FB_RESET : BOOL
END_METHOD

(* ---- L_MC1P_MOTIONUTILS_9400HL.pou ---- *)
FUNCTION_BLOCK L_MC1P_MOTIONUTILS_9400HL EXTENDS L_MC1P_MotionUtils_Base
VAR
	DRIVETYPE : L_MC1P_DriveType;
	GETAXISEXTENSION : L_MC1P_AxisExtensionTypes;
END_VAR
END_FUNCTION_BLOCK

METHOD GETRETAINMEMINFO : L_MC1P_RetainDataType
VAR_OUTPUT
	MEMINFO : L_MC1P_uAxisRetainInfo;
END_VAR
END_METHOD

(* ---- L_MC1P_MOTIONUTILS_9400HL_CAN.pou ---- *)
FUNCTION_BLOCK L_MC1P_MOTIONUTILS_9400HL_CAN EXTENDS L_MC1P_MotionUtils_Base
VAR
	AXISEXTENSION : L_MC1P_AxisExtension_9400HL_CAN;
	DRIVETYPE : L_MC1P_DriveType;
	GETAXISEXTENSION : L_MC1P_AxisExtensionTypes;
END_VAR
END_FUNCTION_BLOCK

(* ---- L_MC1P_MOTIONUTILS_BASE.pou ---- *)
FUNCTION_BLOCK L_MC1P_MOTIONUTILS_BASE
VAR_OUTPUT
	ITFDRIVEUTILS : L_MC1P_IDriveUtils;
END_VAR
VAR
	PDRIVEUTILSCONNECTOR : POINTER TO IoConfigConnector;
	CONNECTEDAXIS : L_IF1P_IFunctionConnection;
	UTILSGUID : L_MC1P_AxisGUID;
	M_ITFEVENTCALLBACK : CmpEventMgr.ICmpEventCallback;
	M_HEVENTUPDATECONFIGURATIONDONE : SysTypes.RTS_IEC_HANDLE;
	M_HINTERFACEUPDATECONFIGURATIONDONE : SysTypes.RTS_IEC_HANDLE;
	_ITFCONNECTSTATUS : L_IF1P_IStatus;
	DRIVETYPE : L_MC1P_DriveType;
	ENCODERTYPE : L_Mc1P_EncoderType;
	GETAXISEXTENSION : L_MC1P_AxisExtensionTypes;
	GETDRIVECONNETOR : POINTER TO IoStandard.IoConfigConnector;
	ITFDEVICECONNECTIONSTATUS : L_IF1P_IStatus;
	NODEGUID : L_MC1P_AxisGUID;
END_VAR
END_FUNCTION_BLOCK

METHOD ACTIVATEAPPCREDITS
VAR_INPUT
	XACTIVATE : BOOL;
END_VAR
END_METHOD

METHOD CALLUPDATECONFIGDONE
END_METHOD

METHOD EVENTCALLBACK : UDINT
VAR_INPUT
	PEVENTPARAM : POINTER TO EventParam;
END_VAR
END_METHOD

METHOD FB_EXIT : BOOL
VAR_INPUT
	BINCOPYCODE : BOOL;
END_VAR
END_METHOD

METHOD GETGUID : BOOL
VAR_INPUT
	PCONNECTOR : POINTER TO IoConfigConnector;
END_VAR
VAR_IN_OUT
	GUID : L_MC1P_AxisGUID;
END_VAR
END_METHOD

METHOD GETMULTIAXISINFO
VAR_IN_OUT
	MULTIAXISINFO : L_MC1P_MultiAxisInfo;
END_VAR
END_METHOD

METHOD GETRETAINMEMINFO : L_MC1P_RetainDataType
VAR_OUTPUT
	MEMINFO : L_MC1P_uAxisRetainInfo;
END_VAR
END_METHOD

METHOD INITSLOTHANDLING : BOOL
VAR_INPUT
	DEVICESLOT : UINT;
END_VAR
END_METHOD

METHOD INITIALIZE : UDINT
VAR_INPUT
	WMODULETYPE : UINT;
	DWINSTANCE : UDINT;
	PCONNECTOR : POINTER TO IoConfigConnector;
END_VAR
END_METHOD

METHOD RESETCONNECTION : L_IE1P_Error
VAR_INPUT
	ITFCALLEDFUNCITON : L_IF1P_IFunctionConnection;
	EDISCONNECTMODE : L_IF1P_DisconnectMode;
	XDISCONNECTEXISTINGCONNECTION : BOOL;
END_VAR
END_METHOD

METHOD SETCONNECTION
VAR_INPUT
	AXISCONNECTION : L_IF1P_IFunctionConnection;
END_VAR
END_METHOD

METHOD FB_INIT : BOOL
VAR_INPUT
	BINITRETAINS : BOOL;
	BINCOPYCODE : BOOL;
END_VAR
END_METHOD

(* ---- L_MC1P_MOTIONUTILS_ENCBPB.pou ---- *)
FUNCTION_BLOCK L_MC1P_MOTIONUTILS_ENCBPB EXTENDS L_MC1P_MotionUtils_Base
VAR
	DRIVETYPE : L_MC1P_DriveType;
	ENCODERTYPE : L_Mc1P_EncoderType;
	GETAXISEXTENSION : L_MC1P_AxisExtensionTypes;
END_VAR
END_FUNCTION_BLOCK

(* ---- L_MC1P_MOTIONUTILS_ENCFREE.pou ---- *)
FUNCTION_BLOCK L_MC1P_MOTIONUTILS_ENCFREE EXTENDS L_MC1P_MotionUtils_Base
VAR
	DRIVETYPE : L_MC1P_DriveType;
	ENCODERTYPE : L_Mc1P_EncoderType;
	GETAXISEXTENSION : L_MC1P_AxisExtensionTypes;
END_VAR
END_FUNCTION_BLOCK

(* ---- L_MC1P_MOTIONUTILS_ENCI500.pou ---- *)
FUNCTION_BLOCK L_MC1P_MOTIONUTILS_ENCI500 EXTENDS L_MC1P_MotionUtils_Base
VAR
	DRIVETYPE : L_MC1P_DriveType;
	ENCODERTYPE : L_Mc1P_EncoderType;
	GETAXISEXTENSION : L_MC1P_AxisExtensionTypes;
END_VAR
END_FUNCTION_BLOCK

(* ---- L_MC1P_MOTIONUTILS_ENCI900_ECAT.pou ---- *)
FUNCTION_BLOCK L_MC1P_MOTIONUTILS_ENCI900_ECAT EXTENDS L_MC1P_MotionUtils_Base
VAR
	DRIVETYPE : L_MC1P_DriveType;
	ENCODERTYPE : L_Mc1P_EncoderType;
	GETAXISEXTENSION : L_MC1P_AxisExtensionTypes;
END_VAR
END_FUNCTION_BLOCK

METHOD GETRETAINMEMINFO : L_MC1P_RetainDataType
VAR_OUTPUT
	MEMINFO : L_MC1P_uAxisRetainInfo;
END_VAR
END_METHOD

(* ---- L_MC1P_MOTIONUTILS_ENCI900_TARGET.pou ---- *)
FUNCTION_BLOCK L_MC1P_MOTIONUTILS_ENCI900_TARGET EXTENDS L_MC1P_MotionUtils_Base
VAR
	DRIVETYPE : L_MC1P_DriveType;
	ENCODERTYPE : L_Mc1P_EncoderType;
	GETAXISEXTENSION : L_MC1P_AxisExtensionTypes;
END_VAR
END_FUNCTION_BLOCK

METHOD GETGUID : BOOL
VAR_INPUT
	PCONNECTOR : POINTER TO IoConfigConnector;
END_VAR
VAR_IN_OUT
	GUID : L_MC1P_AxisGUID;
END_VAR
END_METHOD

METHOD GETRETAINMEMINFO : L_MC1P_RetainDataType
VAR_OUTPUT
	MEMINFO : L_MC1P_uAxisRetainInfo;
END_VAR
END_METHOD

(* ---- L_MC1P_MOTIONUTILS_ENCIOETC.pou ---- *)
FUNCTION_BLOCK L_MC1P_MOTIONUTILS_ENCIOETC EXTENDS L_MC1P_MotionUtils_Base
VAR
	SLICEMODULEHANDLER : L_IMHP_IModuleHandler;
	DRIVETYPE : L_MC1P_DriveType;
	ENCODERTYPE : L_Mc1P_EncoderType;
	GETAXISEXTENSION : L_MC1P_AxisExtensionTypes;
END_VAR
END_FUNCTION_BLOCK

METHOD CALLUPDATECONFIGDONE
END_METHOD

METHOD GETMULTIAXISINFO
VAR_IN_OUT
	MULTIAXISINFO : L_MC1P_MultiAxisInfo;
END_VAR
END_METHOD

(* ---- L_MC1P_MOTIONUTILS_GENERICDRIVE.pou ---- *)
FUNCTION_BLOCK L_MC1P_MOTIONUTILS_GENERICDRIVE EXTENDS L_MC1P_MotionUtils_Base
VAR
	LICHANDLING : L_IMHP_LLMHandling;
	DRIVETYPE : L_MC1P_DriveType;
	GETAXISEXTENSION : L_MC1P_AxisExtensionTypes;
END_VAR
END_FUNCTION_BLOCK

METHOD ACTIVATEAPPCREDITS
VAR_INPUT
	XACTIVATE : BOOL;
END_VAR
END_METHOD

METHOD CALLUPDATECONFIGDONE
END_METHOD

(* ---- L_MC1P_MOTIONUTILS_I500_CAN.pou ---- *)
FUNCTION_BLOCK L_MC1P_MOTIONUTILS_I500_CAN EXTENDS L_MC1P_MotionUtils_Base
VAR
	DRIVETYPE : L_MC1P_DriveType;
	GETAXISEXTENSION : L_MC1P_AxisExtensionTypes;
END_VAR
END_FUNCTION_BLOCK

(* ---- L_MC1P_MOTIONUTILS_I500_ECAT.pou ---- *)
FUNCTION_BLOCK L_MC1P_MOTIONUTILS_I500_ECAT EXTENDS L_MC1P_MotionUtils_Base
VAR
	DRIVETYPE : L_MC1P_DriveType;
	GETAXISEXTENSION : L_MC1P_AxisExtensionTypes;
END_VAR
END_FUNCTION_BLOCK

(* ---- L_MC1P_MOTIONUTILS_I700.pou ---- *)
FUNCTION_BLOCK L_MC1P_MOTIONUTILS_I700 EXTENDS L_MC1P_MotionUtils_Base
VAR_INPUT
	PCONNECTORFORMULTIAXISHANDLING : POINTER TO IoConfigConnector;
END_VAR
VAR
	UISLOT : UINT;
	ITFSLAVEAXISMODULEHANDLER : L_IMHP_IModuleHandler;
	SLAVEMULTIAXISMODULEHANDLERBASE : L_IMHP_ModuleHandler := STRUCT(SuspendRegistration := TRUE, UseLEM := TRUE, Layer := L_IMHP_Layer.Communication, CompType := L_IMHP_ComponentType.EtherCATSlave, DefaultRelationShip := L_IMHP_RelationshipID.CommunicationView);
	DRIVETYPE : L_MC1P_DriveType;
	GETAXISEXTENSION : L_MC1P_AxisExtensionTypes;
END_VAR
END_FUNCTION_BLOCK

METHOD CALLUPDATECONFIGDONE
END_METHOD

METHOD GETMULTIAXISINFO
VAR_IN_OUT
	MULTIAXISINFO : L_MC1P_MultiAxisInfo;
END_VAR
END_METHOD

METHOD GETRETAINMEMINFO : L_MC1P_RetainDataType
VAR_OUTPUT
	MEMINFO : L_MC1P_uAxisRetainInfo;
END_VAR
END_METHOD

METHOD INITSLOTHANDLING : BOOL
VAR_INPUT
	DEVICESLOT : UINT;
END_VAR
END_METHOD
